LIN {X 0,Y 354.829,Z 449.908,A -85,B 0,C 180,E1 -13477.894,E2 -13477.894} C_VEL
LIN {X 0,Y 354.917,Z 449.897,A -85,B 0,C 180,E1 -13481.892,E2 -13481.892} C_VEL
LIN {X 0,Y 354.937,Z 449.895,A -85,B 0,C 180,E1 -13485.981,E2 -13485.981} C_VEL
LIN {X 0,Y 354.973,Z 449.891,A -85,B 0,C 180,E1 -13489.736,E2 -13489.736} C_VEL
LIN {X 0,Y 355.108,Z 449.874,A -85,B 0,C 180,E1 -13492.037,E2 -13492.037} C_VEL
LIN {X 0,Y 355.087,Z 449.879,A -85,B 0,C 180,E1 -13494.321,E2 -13494.321} C_VEL
LIN {X 0,Y 355.241,Z 449.857,A -85,B 0,C 180,E1 -13497.733,E2 -13497.733} C_VEL
LIN {X 0,Y 355.392,Z 449.839,A -85,B 0,C 180,E1 -13500,E2 -13500} C_VEL
LIN {X 0,Y 355.241,Z 449.86,A -85,B 0,C 180,E1 -13502.268,E2 -13502.268} C_VEL
LIN {X 0,Y 355.137,Z 449.873,A -85,B 0,C 180,E1 -13506.819,E2 -13506.819} C_VEL
LIN {X 0,Y 355.01,Z 449.887,A -85,B 0,C 180,E1 -13509.113,E2 -13509.113} C_VEL
LIN {X 0,Y 354.916,Z 449.902,A -85,B 0,C 180,E1 -13512.581,E2 -13512.581} C_VEL
LIN {X 0,Y 354.884,Z 449.905,A -85,B 0,C 180,E1 -13516.096,E2 -13516.096} C_VEL
LIN {X 0,Y 354.902,Z 449.904,A -85,B 0,C 180,E1 -13518.472,E2 -13518.472} C_VEL
LIN {X 0,Y 354.83,Z 449.912,A -85,B 0,C 180,E1 -13522.107,E2 -13522.107} C_VEL
LIN {X 0,Y 354.895,Z 449.903,A -85,B 0,C 180,E1 -13525.828,E2 -13525.828} C_VEL
LIN {X 0,Y 354.85,Z 449.907,A -85,B 0,C 180,E1 -13529.679,E2 -13529.679} C_VEL
LIN {X 0,Y 354.803,Z 449.914,A -85,B 0,C 180,E1 -13533.703,E2 -13533.703} C_VEL
LIN {X 0,Y 354.796,Z 449.915,A -85,B 0,C 180,E1 -13536.46,E2 -13536.46} C_VEL
LIN {X 0,Y 354.822,Z 449.91,A -85,B 0,C 180,E1 -13539.424,E2 -13539.424} C_VEL
LIN {X 0,Y 354.787,Z 449.914,A -85,B 0,C 180,E1 -13542.868,E2 -13542.868} C_VEL
LIN {X 0,Y 354.775,Z 449.92,A -85,B 0,C 180,E1 -13546.106,E2 -13546.106} C_VEL
LIN {X 0,Y 354.824,Z 449.909,A -85,B 0,C 180,E1 -13549.185,E2 -13549.185} C_VEL
LIN {X 0,Y 354.809,Z 449.913,A -85,B 0,C 180,E1 -13552.403,E2 -13552.403} C_VEL
LIN {X 0,Y 354.813,Z 449.91,A -85,B 0,C 180,E1 -13554.942,E2 -13554.942} C_VEL
LIN {X 0,Y 354.795,Z 449.914,A -85,B 0,C 180,E1 -13558.406,E2 -13558.406} C_VEL
LIN {X 0,Y 354.855,Z 449.91,A -85,B 0,C 180,E1 -13561.62,E2 -13561.62} C_VEL
LIN {X 0,Y 354.901,Z 449.902,A -85,B 0,C 180,E1 -13564.173,E2 -13564.173} C_VEL
LIN {X 0,Y 354.837,Z 449.911,A -85,B 0,C 180,E1 -13567.895,E2 -13567.895} C_VEL
LIN {X 0,Y 354.926,Z 449.9,A -85,B 0,C 180,E1 -13571.892,E2 -13571.892} C_VEL
LIN {X 0,Y 354.946,Z 449.896,A -85,B 0,C 180,E1 -13575.981,E2 -13575.981} C_VEL
LIN {X 0,Y 354.981,Z 449.894,A -85,B 0,C 180,E1 -13579.736,E2 -13579.736} C_VEL
LIN {X 0,Y 355.103,Z 449.878,A -85,B 0,C 180,E1 -13583.18,E2 -13583.18} C_VEL
LIN {X 0,Y 355.249,Z 449.859,A -85,B 0,C 180,E1 -13587.732,E2 -13587.732} C_VEL
LIN {X 0,Y 355.4,Z 449.838,A -85,B 0,C 180,E1 -13590,E2 -13590} C_VEL
LIN {X 0,Y 355.248,Z 449.857,A -85,B 0,C 180,E1 -13592.268,E2 -13592.268} C_VEL
LIN {X 0,Y 355.126,Z 449.873,A -85,B 0,C 180,E1 -13596.819,E2 -13596.819} C_VEL
LIN {X 0,Y 354.981,Z 449.889,A -85,B 0,C 180,E1 -13600.264,E2 -13600.264} C_VEL
LIN {X 0,Y 354.946,Z 449.894,A -85,B 0,C 180,E1 -13604.019,E2 -13604.019} C_VEL
LIN {X 0,Y 354.925,Z 449.896,A -85,B 0,C 180,E1 -13608.108,E2 -13608.108} C_VEL
LIN {X 0,Y 354.837,Z 449.907,A -85,B 0,C 180,E1 -13612.105,E2 -13612.105} C_VEL
LIN {X 0,Y 354.901,Z 449.9,A -85,B 0,C 180,E1 -13615.827,E2 -13615.827} C_VEL
LIN {X 0,Y 354.855,Z 449.906,A -85,B 0,C 180,E1 -13619.678,E2 -13619.678} C_VEL
LIN {X 0,Y 354.779,Z 449.915,A -85,B 0,C 180,E1 -13623.695,E2 -13623.695} C_VEL
LIN {X 0,Y 354.538,Z 449.947,A -85,B 0,C 180,E1 -13626.49,E2 -13626.49} C_VEL
LIN {X 0,Y 354.177,Z 449.995,A -85,B 0,C 180,E1 -13629.418,E2 -13629.418} C_VEL
LIN {X 0,Y 353.996,Z 450.018,A -85,B 0,C 180,E1 -13631.024,E2 -13631.024} C_VEL
LIN {X 0,Y 353.844,Z 450.744,A -85,B 0,C 180,E1 -13632.702,E2 -13632.702} C_VEL
LIN {X 0,Y 353.757,Z 453.469,A -85,B 0,C 180,E1 -13635.946,E2 -13635.946} C_VEL
LIN {X 0,Y 353.742,Z 455.553,A -85,B 0,C 180,E1 -13638.16,E2 -13638.16} C_VEL
LIN {X 0,Y 358.097,Z 470.69,A -85,B 0,C 180,E1 -13639.011,E2 -13639.011} C_VEL
LIN {X 0,Y 361.351,Z 483.198,A -85,B 0,C 180,E1 -13639.883,E2 -13639.883} C_VEL
LIN {X 0,Y 361.484,Z 485.632,A -85,B 0,C 180,E1 -13640.044,E2 -13640.044} C_VEL
LIN {X 0,Y 360.572,Z 489.26,A -85,B 0,C 180,E1 -13640.246,E2 -13640.246} C_VEL
LIN {X 0,Y 355.882,Z 498.667,A -85,B 0,C 180,E1 -13640.734,E2 -13640.734} C_VEL
LIN {X 0,Y 354.987,Z 502.273,A -85,B 0,C 180,E1 -13641.006,E2 -13641.006} C_VEL
LIN {X 0,Y 353.73,Z 515.023,A -85,B 0,C 180,E1 -13642.22,E2 -13642.22} C_VEL
LIN {X 0,Y 352.398,Z 526.861,A -85,B 0,C 180,E1 -13643.607,E2 -13643.607} C_VEL
LIN {X 0,Y 351.136,Z 537.648,A -85,B 0,C 180,E1 -13645.145,E2 -13645.145} C_VEL
LIN {X 0,Y 349.979,Z 547.411,A -85,B 0,C 180,E1 -13646.824,E2 -13646.824} C_VEL
LIN {X 0,Y 348.764,Z 556.624,A -85,B 0,C 180,E1 -13648.742,E2 -13648.742} C_VEL
LIN {X 0,Y 347.986,Z 563.988,A -85,B 0,C 180,E1 -13650.618,E2 -13650.618} C_VEL
LIN {X 0,Y 347.432,Z 569.383,A -85,B 0,C 180,E1 -13652.273,E2 -13652.273} C_VEL
LIN {X 0,Y 346.933,Z 574.46,A -85,B 0,C 180,E1 -13654.18,E2 -13654.18} C_VEL
LIN {X 0,Y 346.575,Z 578.385,A -85,B 0,C 180,E1 -13656.073,E2 -13656.073} C_VEL
LIN {X 0,Y 346.371,Z 580.441,A -85,B 0,C 180,E1 -13657.324,E2 -13657.324} C_VEL
LIN {X 0,Y 346.25,Z 582.506,A -85,B 0,C 180,E1 -13659.014,E2 -13659.014} C_VEL
LIN {X 0,Y 346.14,Z 584.057,A -85,B 0,C 180,E1 -13661.042,E2 -13661.042} C_VEL
LIN {X 0,Y 346.193,Z 584.56,A -85,B 0,C 180,E1 -13662.577,E2 -13662.577} C_VEL
LIN {X 0,Y 346.282,Z 584.255,A -85,B 0,C 180,E1 -13664.701,E2 -13664.701} C_VEL
LIN {X 0,Y 346.641,Z 582.569,A -85,B 0,C 180,E1 -13667.113,E2 -13667.113} C_VEL
LIN {X 0,Y 347.177,Z 579.418,A -85,B 0,C 180,E1 -13669.502,E2 -13669.502} C_VEL
LIN {X 0,Y 347.95,Z 574.76,A -85,B 0,C 180,E1 -13671.872,E2 -13671.872} C_VEL
LIN {X 0,Y 349.05,Z 568.481,A -85,B 0,C 180,E1 -13674.222,E2 -13674.222} C_VEL
LIN {X 0,Y 350.323,Z 561.496,A -85,B 0,C 180,E1 -13676.261,E2 -13676.261} C_VEL
LIN {X 0,Y 351.606,Z 554.204,A -85,B 0,C 180,E1 -13678.007,E2 -13678.007} C_VEL
LIN {X 0,Y 353.21,Z 545.579,A -85,B 0,C 180,E1 -13679.715,E2 -13679.715} C_VEL
LIN {X 0,Y 355.07,Z 535.172,A -85,B 0,C 180,E1 -13681.418,E2 -13681.418} C_VEL
LIN {X 0,Y 356.945,Z 523.616,A -85,B 0,C 180,E1 -13682.962,E2 -13682.962} C_VEL
LIN {X 0,Y 358.844,Z 510.865,A -85,B 0,C 180,E1 -13684.352,E2 -13684.352} C_VEL
LIN {X 0,Y 360.62,Z 497.644,A -85,B 0,C 180,E1 -13685.503,E2 -13685.503} C_VEL
LIN {X 0,Y 360.499,Z 495.401,A -85,B 0,C 180,E1 -13685.715,E2 -13685.715} C_VEL
LIN {X 0,Y 356.948,Z 482.251,A -85,B 0,C 180,E1 -13687.113,E2 -13687.113} C_VEL
LIN {X 0,Y 352.491,Z 471.337,A -85,B 0,C 180,E1 -13688.319,E2 -13688.319} C_VEL
LIN {X 0,Y 349.273,Z 464.852,A -85,B 0,C 180,E1 -13689.061,E2 -13689.061} C_VEL
LIN {X 0,Y 348.009,Z 462.121,A -85,B 0,C 180,E1 -13689.352,E2 -13689.352} C_VEL
LIN {X 0,Y 347.894,Z 461.481,A -85,B 0,C 180,E1 -13689.447,E2 -13689.447} C_VEL
LIN {X 0,Y 348.089,Z 459.823,A -85,B 0,C 180,E1 -13692.832,E2 -13692.832} C_VEL
LIN {X 0,Y 348.261,Z 458.785,A -85,B 0,C 180,E1 -13695.209,E2 -13695.209} C_VEL
LIN {X 0,Y 348.561,Z 457.476,A -85,B 0,C 180,E1 -13698.82,E2 -13698.82} C_VEL
LIN {X 0,Y 348.633,Z 456.533,A -85,B 0,C 180,E1 -13702.52,E2 -13702.52} C_VEL
LIN {X 0,Y 348.681,Z 456.169,A -85,B 0,C 180,E1 -13705.041,E2 -13705.041} C_VEL
LIN {X 0,Y 348.679,Z 456.038,A -85,B 0,C 180,E1 -13707.619,E2 -13707.619} C_VEL
LIN {X 0,Y 348.7,Z 456.207,A -85,B 0,C 180,E1 -13710.256,E2 -13710.256} C_VEL
LIN {X 0,Y 348.809,Z 456.707,A -85,B 0,C 180,E1 -13712.957,E2 -13712.957} C_VEL
LIN {X 0,Y 348.995,Z 457.843,A -85,B 0,C 180,E1 -13716.342,E2 -13716.342} C_VEL
LIN {X 0,Y 349.394,Z 459.832,A -85,B 0,C 180,E1 -13720.151,E2 -13720.151} C_VEL
LIN {X 0,Y 349.843,Z 462.423,A -85,B 0,C 180,E1 -13723.681,E2 -13723.681} C_VEL
LIN {X 0,Y 350.325,Z 465.525,A -85,B 0,C 180,E1 -13726.994,E2 -13726.994} C_VEL
LIN {X 0,Y 350.645,Z 468.414,A -85,B 0,C 180,E1 -13729.608,E2 -13729.608} C_VEL
LIN {X 0,Y 350.514,Z 470.912,A -85,B 0,C 180,E1 -13731.57,E2 -13731.57} C_VEL
LIN {X 0,Y 349.85,Z 474.877,A -85,B 0,C 180,E1 -13734.369,E2 -13734.369} C_VEL
LIN {X 0,Y 349.012,Z 480.13,A -85,B 0,C 180,E1 -13737.752,E2 -13737.752} C_VEL
LIN {X 0,Y 348.283,Z 485.659,A -85,B 0,C 180,E1 -13741.034,E2 -13741.034} C_VEL
LIN {X 0,Y 347.988,Z 488.32,A -85,B 0,C 180,E1 -13742.549,E2 -13742.549} C_VEL
LIN {X 0,Y 348.94,Z 491.893,A -85,B 0,C 180,E1 -13742.833,E2 -13742.833} C_VEL
LIN {X 0,Y 352.14,Z 502.047,A -85,B 0,C 180,E1 -13743.686,E2 -13743.686} C_VEL
LIN {X 0,Y 355.247,Z 515.449,A -85,B 0,C 180,E1 -13744.835,E2 -13744.835} C_VEL
LIN {X 0,Y 356.989,Z 529.251,A -85,B 0,C 180,E1 -13746.039,E2 -13746.039} C_VEL
LIN {X 0,Y 357.339,Z 542.457,A -85,B 0,C 180,E1 -13747.296,E2 -13747.296} C_VEL
LIN {X 0,Y 355.2,Z 556.001,A -85,B 0,C 180,E1 -13748.646,E2 -13748.646} C_VEL
LIN {X 0,Y 353.175,Z 568.787,A -85,B 0,C 180,E1 -13750.228,E2 -13750.228} C_VEL
LIN {X 0,Y 351.295,Z 580.082,A -85,B 0,C 180,E1 -13751.936,E2 -13751.936} C_VEL
LIN {X 0,Y 349.771,Z 589.495,A -85,B 0,C 180,E1 -13753.662,E2 -13753.662} C_VEL
LIN {X 0,Y 348.467,Z 598.551,A -85,B 0,C 180,E1 -13755.672,E2 -13755.672} C_VEL
LIN {X 0,Y 347.475,Z 606.146,A -85,B 0,C 180,E1 -13757.739,E2 -13757.739} C_VEL
LIN {X 0,Y 346.705,Z 612.966,A -85,B 0,C 180,E1 -13760.078,E2 -13760.078} C_VEL
LIN {X 0,Y 346.371,Z 618.146,A -85,B 0,C 180,E1 -13762.421,E2 -13762.421} C_VEL
LIN {X 0,Y 346.248,Z 621.01,A -85,B 0,C 180,E1 -13764.175,E2 -13764.175} C_VEL
LIN {X 0,Y 346.219,Z 623.573,A -85,B 0,C 180,E1 -13766.509,E2 -13766.509} C_VEL
LIN {X 0,Y 346.4,Z 624.733,A -85,B 0,C 180,E1 -13768.837,E2 -13768.837} C_VEL
LIN {X 0,Y 346.41,Z 624.472,A -85,B 0,C 180,E1 -13771.162,E2 -13771.162} C_VEL
LIN {X 0,Y 346.231,Z 622.778,A -85,B 0,C 180,E1 -13773.491,E2 -13773.491} C_VEL
LIN {X 0,Y 346.3,Z 621.398,A -85,B 0,C 180,E1 -13774.656,E2 -13774.656} C_VEL
LIN {X 0,Y 346.366,Z 617.463,A -85,B 0,C 180,E1 -13776.993,E2 -13776.993} C_VEL
LIN {X 0,Y 346.609,Z 611.869,A -85,B 0,C 180,E1 -13779.335,E2 -13779.335} C_VEL
LIN {X 0,Y 347.095,Z 605.516,A -85,B 0,C 180,E1 -13781.386,E2 -13781.386} C_VEL
LIN {X 0,Y 347.902,Z 597.587,A -85,B 0,C 180,E1 -13783.433,E2 -13783.433} C_VEL
LIN {X 0,Y 348.598,Z 590.314,A -85,B 0,C 180,E1 -13784.988,E2 -13784.988} C_VEL
LIN {X 0,Y 349.659,Z 581.104,A -85,B 0,C 180,E1 -13786.643,E2 -13786.643} C_VEL
LIN {X 0,Y 350.922,Z 570.429,A -85,B 0,C 180,E1 -13788.235,E2 -13788.235} C_VEL
LIN {X 0,Y 352.268,Z 560.02,A -85,B 0,C 180,E1 -13789.522,E2 -13789.522} C_VEL
LIN {X 0,Y 353.719,Z 547.45,A -85,B 0,C 180,E1 -13790.803,E2 -13790.803} C_VEL
LIN {X 0,Y 354.551,Z 539.176,A -85,B 0,C 180,E1 -13791.512,E2 -13791.512} C_VEL
LIN {X 0,Y 353.044,Z 526.06,A -85,B 0,C 180,E1 -13792.554,E2 -13792.554} C_VEL
LIN {X 0,Y 350.623,Z 511.086,A -85,B 0,C 180,E1 -13793.529,E2 -13793.529} C_VEL
LIN {X 0,Y 347.827,Z 495.803,A -85,B 0,C 180,E1 -13794.297,E2 -13794.297} C_VEL
LIN {X 0,Y 347.476,Z 493.605,A -85,B 0,C 180,E1 -13794.412,E2 -13794.412} C_VEL
LIN {X 0,Y 348.026,Z 487.442,A -85,B 0,C 180,E1 -13797.675,E2 -13797.675} C_VEL
LIN {X 0,Y 348.651,Z 481.404,A -85,B 0,C 180,E1 -13800.931,E2 -13800.931} C_VEL
LIN {X 0,Y 349.401,Z 475.058,A -85,B 0,C 180,E1 -13804.443,E2 -13804.443} C_VEL
LIN {X 0,Y 350.106,Z 469.257,A -85,B 0,C 180,E1 -13807.752,E2 -13807.752} C_VEL
LIN {X 0,Y 350.303,Z 465.561,A -85,B 0,C 180,E1 -13809.941,E2 -13809.941} C_VEL
LIN {X 0,Y 349.553,Z 460.534,A -85,B 0,C 180,E1 -13813.124,E2 -13813.124} C_VEL
LIN {X 0,Y 348.571,Z 455.182,A -85,B 0,C 180,E1 -13816.724,E2 -13816.724} C_VEL
LIN {X 0,Y 347.827,Z 450.784,A -85,B 0,C 180,E1 -13819.854,E2 -13819.854} C_VEL
LIN {X 0,Y 347.766,Z 450.788,A -85,B 0,C 180,E1 -13823.935,E2 -13823.935} C_VEL
LIN {X 0,Y 347.743,Z 450.796,A -85,B 0,C 180,E1 -13826.929,E2 -13826.929} C_VEL
LIN {X 0,Y 347.802,Z 450.789,A -85,B 0,C 180,E1 -13830.99,E2 -13830.99} C_VEL
LIN {X 0,Y 347.827,Z 450.781,A -85,B 0,C 180,E1 -13833.608,E2 -13833.608} C_VEL
LIN {X 0,Y 347.783,Z 450.786,A -85,B 0,C 180,E1 -13836.162,E2 -13836.162} C_VEL
LIN {X 0,Y 347.807,Z 450.783,A -85,B 0,C 180,E1 -13839.909,E2 -13839.909} C_VEL
LIN {X 0,Y 347.861,Z 450.778,A -85,B 0,C 180,E1 -13842.359,E2 -13842.359} C_VEL
LIN {X 0,Y 347.892,Z 450.772,A -85,B 0,C 180,E1 -13845.971,E2 -13845.971} C_VEL
LIN {X 0,Y 347.923,Z 450.769,A -85,B 0,C 180,E1 -13849.526,E2 -13849.526} C_VEL
LIN {X 0,Y 348.068,Z 450.751,A -85,B 0,C 180,E1 -13851.875,E2 -13851.875} C_VEL
LIN {X 0,Y 348.062,Z 450.753,A -85,B 0,C 180,E1 -13854.206,E2 -13854.206} C_VEL
LIN {X 0,Y 348.203,Z 450.734,A -85,B 0,C 180,E1 -13857.687,E2 -13857.687} C_VEL
LIN {X 0,Y 348.34,Z 450.717,A -85,B 0,C 180,E1 -13860,E2 -13860} C_VEL
LIN {X 0,Y 348.203,Z 450.737,A -85,B 0,C 180,E1 -13862.314,E2 -13862.314} C_VEL
LIN {X 0,Y 348.104,Z 450.748,A -85,B 0,C 180,E1 -13866.958,E2 -13866.958} C_VEL
LIN {X 0,Y 347.962,Z 450.764,A -85,B 0,C 180,E1 -13869.299,E2 -13869.299} C_VEL
LIN {X 0,Y 347.885,Z 450.775,A -85,B 0,C 180,E1 -13872.84,E2 -13872.84} C_VEL
LIN {X 0,Y 347.834,Z 450.785,A -85,B 0,C 180,E1 -13876.432,E2 -13876.432} C_VEL
LIN {X 0,Y 347.851,Z 450.779,A -85,B 0,C 180,E1 -13878.861,E2 -13878.861} C_VEL
LIN {X 0,Y 347.77,Z 450.791,A -85,B 0,C 180,E1 -13882.58,E2 -13882.58} C_VEL
LIN {X 0,Y 347.808,Z 450.783,A -85,B 0,C 180,E1 -13885.109,E2 -13885.109} C_VEL
LIN {X 0,Y 347.806,Z 450.784,A -85,B 0,C 180,E1 -13887.695,E2 -13887.695} C_VEL
LIN {X 0,Y 347.76,Z 450.793,A -85,B 0,C 180,E1 -13890.347,E2 -13890.347} C_VEL
LIN {X 0,Y 347.741,Z 450.794,A -85,B 0,C 180,E1 -13894.465,E2 -13894.465} C_VEL
LIN {X 0,Y 347.772,Z 450.793,A -85,B 0,C 180,E1 -13897.99,E2 -13897.99} C_VEL
LIN {X 0,Y 347.749,Z 450.794,A -85,B 0,C 180,E1 -13901.831,E2 -13901.831} C_VEL
LIN {X 0,Y 347.707,Z 450.795,A -85,B 0,C 180,E1 -13905.027,E2 -13905.027} C_VEL
LIN {X 0,Y 347.767,Z 450.79,A -85,B 0,C 180,E1 -13908.395,E2 -13908.395} C_VEL
LIN {X 0,Y 347.776,Z 450.792,A -85,B 0,C 180,E1 -13912.012,E2 -13912.012} C_VEL
LIN {X 0,Y 347.745,Z 450.794,A -85,B 0,C 180,E1 -13915.537,E2 -13915.537} C_VEL
LIN {X 0,Y 347.765,Z 450.793,A -85,B 0,C 180,E1 -13919.654,E2 -13919.654} C_VEL
LIN {X 0,Y 347.854,Z 450.777,A -85,B 0,C 180,E1 -13922.745,E2 -13922.745} C_VEL
LIN {X 0,Y 347.791,Z 450.787,A -85,B 0,C 180,E1 -13926.163,E2 -13926.163} C_VEL
LIN {X 0,Y 347.82,Z 450.785,A -85,B 0,C 180,E1 -13929.91,E2 -13929.91} C_VEL
LIN {X 0,Y 347.869,Z 450.776,A -85,B 0,C 180,E1 -13932.36,E2 -13932.36} C_VEL
LIN {X 0,Y 347.9,Z 450.773,A -85,B 0,C 180,E1 -13935.971,E2 -13935.971} C_VEL
LIN {X 0,Y 347.932,Z 450.773,A -85,B 0,C 180,E1 -13939.526,E2 -13939.526} C_VEL
LIN {X 0,Y 348.071,Z 450.752,A -85,B 0,C 180,E1 -13943.042,E2 -13943.042} C_VEL
LIN {X 0,Y 348.211,Z 450.736,A -85,B 0,C 180,E1 -13947.687,E2 -13947.687} C_VEL
LIN {X 0,Y 348.349,Z 450.716,A -85,B 0,C 180,E1 -13950,E2 -13950} C_VEL
LIN {X 0,Y 348.21,Z 450.733,A -85,B 0,C 180,E1 -13952.313,E2 -13952.313} C_VEL
LIN {X 0,Y 348.092,Z 450.75,A -85,B 0,C 180,E1 -13956.958,E2 -13956.958} C_VEL
LIN {X 0,Y 347.932,Z 450.768,A -85,B 0,C 180,E1 -13960.474,E2 -13960.474} C_VEL
LIN {X 0,Y 347.901,Z 450.771,A -85,B 0,C 180,E1 -13964.149,E2 -13964.149} C_VEL
LIN {X 0,Y 347.893,Z 450.772,A -85,B 0,C 180,E1 -13968.29,E2 -13968.29} C_VEL
LIN {X 0,Y 347.791,Z 450.786,A -85,B 0,C 180,E1 -13971.635,E2 -13971.635} C_VEL
LIN {X 0,Y 347.815,Z 450.787,A -85,B 0,C 180,E1 -13975.108,E2 -13975.108} C_VEL
LIN {X 0,Y 347.811,Z 450.783,A -85,B 0,C 180,E1 -13977.693,E2 -13977.693} C_VEL
LIN {X 0,Y 347.764,Z 450.789,A -85,B 0,C 180,E1 -13980.346,E2 -13980.346} C_VEL
LIN {X 0,Y 347.712,Z 450.795,A -85,B 0,C 180,E1 -13984.034,E2 -13984.034} C_VEL
LIN {X 0,Y 347.383,Z 450.838,A -85,B 0,C 180,E1 -13987.368,E2 -13987.368} C_VEL
LIN {X 0,Y 347.013,Z 450.888,A -85,B 0,C 180,E1 -13990.397,E2 -13990.397} C_VEL
LIN {X 0,Y 346.799,Z 450.914,A -85,B 0,C 180,E1 -13991.97,E2 -13991.97} C_VEL
LIN {X 0,Y 346.719,Z 453.556,A -85,B 0,C 180,E1 -13995.189,E2 -13995.189} C_VEL
LIN {X 0,Y 346.668,Z 455.811,A -85,B 0,C 180,E1 -13997.751,E2 -13997.751} C_VEL
LIN {X 0,Y 350.723,Z 469.912,A -85,B 0,C 180,E1 -13998.56,E2 -13998.56} C_VEL
LIN {X 0,Y 354.542,Z 484.531,A -85,B 0,C 180,E1 -13999.604,E2 -13999.604} C_VEL
LIN {X 0,Y 355.941,Z 491.589,A -85,B 0,C 180,E1 -14000.172,E2 -14000.172} C_VEL
LIN {X 0,Y 354.987,Z 502.273,A -85,B 0,C 180,E1 -14001.006,E2 -14001.006} C_VEL
LIN {X 0,Y 353.88,Z 507.456,A -85,B 0,C 180,E1 -14001.429,E2 -14001.429} C_VEL
LIN {X 0,Y 350.294,Z 515.693,A -85,B 0,C 180,E1 -14002.113,E2 -14002.113} C_VEL
LIN {X 0,Y 346.615,Z 523.574,A -85,B 0,C 180,E1 -14002.897,E2 -14002.897} C_VEL
LIN {X 0,Y 345.377,Z 528.2,A -85,B 0,C 180,E1 -14003.471,E2 -14003.471} C_VEL
LIN {X 0,Y 344.049,Z 539.278,A -85,B 0,C 180,E1 -14005.112,E2 -14005.112} C_VEL
LIN {X 0,Y 342.845,Z 549.219,A -85,B 0,C 180,E1 -14006.898,E2 -14006.898} C_VEL
LIN {X 0,Y 341.687,Z 557.596,A -85,B 0,C 180,E1 -14008.711,E2 -14008.711} C_VEL
LIN {X 0,Y 340.884,Z 565.063,A -85,B 0,C 180,E1 -14010.682,E2 -14010.682} C_VEL
LIN {X 0,Y 340.128,Z 571.996,A -85,B 0,C 180,E1 -14012.962,E2 -14012.962} C_VEL
LIN {X 0,Y 339.709,Z 576.583,A -85,B 0,C 180,E1 -14014.905,E2 -14014.905} C_VEL
LIN {X 0,Y 339.349,Z 580.082,A -85,B 0,C 180,E1 -14016.828,E2 -14016.828} C_VEL
LIN {X 0,Y 339.174,Z 582.694,A -85,B 0,C 180,E1 -14018.816,E2 -14018.816} C_VEL
LIN {X 0,Y 339.079,Z 584.251,A -85,B 0,C 180,E1 -14020.632,E2 -14020.632} C_VEL
LIN {X 0,Y 339.101,Z 585.029,A -85,B 0,C 180,E1 -14023.132,E2 -14023.132} C_VEL
LIN {X 0,Y 339.319,Z 584.338,A -85,B 0,C 180,E1 -14025.608,E2 -14025.608} C_VEL
LIN {X 0,Y 339.743,Z 582.218,A -85,B 0,C 180,E1 -14028.061,E2 -14028.061} C_VEL
LIN {X 0,Y 340.421,Z 578.652,A -85,B 0,C 180,E1 -14030.493,E2 -14030.493} C_VEL
LIN {X 0,Y 341.086,Z 574.873,A -85,B 0,C 180,E1 -14032.338,E2 -14032.338} C_VEL
LIN {X 0,Y 342.308,Z 568.637,A -85,B 0,C 180,E1 -14034.699,E2 -14034.699} C_VEL
LIN {X 0,Y 343.717,Z 561.604,A -85,B 0,C 180,E1 -14036.776,E2 -14036.776} C_VEL
LIN {X 0,Y 345.32,Z 552.941,A -85,B 0,C 180,E1 -14038.834,E2 -14038.834} C_VEL
LIN {X 0,Y 347.108,Z 543.891,A -85,B 0,C 180,E1 -14040.58,E2 -14040.58} C_VEL
LIN {X 0,Y 349.117,Z 533.081,A -85,B 0,C 180,E1 -14042.307,E2 -14042.307} C_VEL
LIN {X 0,Y 351.19,Z 521.065,A -85,B 0,C 180,E1 -14043.873,E2 -14043.873} C_VEL
LIN {X 0,Y 353.203,Z 508.147,A -85,B 0,C 180,E1 -14045.23,E2 -14045.23} C_VEL
LIN {X 0,Y 354.445,Z 498.262,A -85,B 0,C 180,E1 -14046.088,E2 -14046.088} C_VEL
LIN {X 0,Y 351.256,Z 485.636,A -85,B 0,C 180,E1 -14047.523,E2 -14047.523} C_VEL
LIN {X 0,Y 346.264,Z 473.099,A -85,B 0,C 180,E1 -14049,E2 -14049} C_VEL
LIN {X 0,Y 342.347,Z 465.595,A -85,B 0,C 180,E1 -14049.94,E2 -14049.94} C_VEL
LIN {X 0,Y 341.095,Z 462.937,A -85,B 0,C 180,E1 -14050.248,E2 -14050.248} C_VEL
LIN {X 0,Y 340.973,Z 462.196,A -85,B 0,C 180,E1 -14050.352,E2 -14050.352} C_VEL
LIN {X 0,Y 341.251,Z 460.309,A -85,B 0,C 180,E1 -14054.548,E2 -14054.548} C_VEL
LIN {X 0,Y 341.607,Z 458.778,A -85,B 0,C 180,E1 -14058.852,E2 -14058.852} C_VEL
LIN {X 0,Y 341.683,Z 457.983,A -85,B 0,C 180,E1 -14062.244,E2 -14062.244} C_VEL
LIN {X 0,Y 341.711,Z 457.556,A -85,B 0,C 180,E1 -14065.589,E2 -14065.589} C_VEL
LIN {X 0,Y 341.714,Z 457.546,A -85,B 0,C 180,E1 -14068.232,E2 -14068.232} C_VEL
LIN {X 0,Y 341.762,Z 457.817,A -85,B 0,C 180,E1 -14070.937,E2 -14070.937} C_VEL
LIN {X 0,Y 341.878,Z 458.436,A -85,B 0,C 180,E1 -14073.713,E2 -14073.713} C_VEL
LIN {X 0,Y 342.1,Z 459.568,A -85,B 0,C 180,E1 -14076.756,E2 -14076.756} C_VEL
LIN {X 0,Y 342.385,Z 460.999,A -85,B 0,C 180,E1 -14079.518,E2 -14079.518} C_VEL
LIN {X 0,Y 342.772,Z 463.057,A -85,B 0,C 180,E1 -14082.579,E2 -14082.579} C_VEL
LIN {X 0,Y 343.214,Z 465.864,A -85,B 0,C 180,E1 -14085.877,E2 -14085.877} C_VEL
LIN {X 0,Y 343.474,Z 467.495,A -85,B 0,C 180,E1 -14087.529,E2 -14087.529} C_VEL
LIN {X 0,Y 343.636,Z 469.296,A -85,B 0,C 180,E1 -14089.176,E2 -14089.176} C_VEL
LIN {X 0,Y 343.405,Z 472.97,A -85,B 0,C 180,E1 -14092.124,E2 -14092.124} C_VEL
LIN {X 0,Y 342.658,Z 477.228,A -85,B 0,C 180,E1 -14095.126,E2 -14095.126} C_VEL
LIN {X 0,Y 341.713,Z 483.346,A -85,B 0,C 180,E1 -14099.058,E2 -14099.058} C_VEL
LIN {X 0,Y 341.159,Z 487.68,A -85,B 0,C 180,E1 -14101.656,E2 -14101.656} C_VEL
LIN {X 0,Y 342.044,Z 491.064,A -85,B 0,C 180,E1 -14101.929,E2 -14101.929} C_VEL
LIN {X 0,Y 345.422,Z 501.575,A -85,B 0,C 180,E1 -14102.895,E2 -14102.895} C_VEL
LIN {X 0,Y 348.64,Z 514.814,A -85,B 0,C 180,E1 -14104.102,E2 -14104.102} C_VEL
LIN {X 0,Y 350.333,Z 527.227,A -85,B 0,C 180,E1 -14105.253,E2 -14105.253} C_VEL
LIN {X 0,Y 350.875,Z 538.928,A -85,B 0,C 180,E1 -14106.385,E2 -14106.385} C_VEL
LIN {X 0,Y 350.632,Z 544.943,A -85,B 0,C 180,E1 -14106.993,E2 -14106.993} C_VEL
LIN {X 0,Y 348.605,Z 556.949,A -85,B 0,C 180,E1 -14108.256,E2 -14108.256} C_VEL
LIN {X 0,Y 346.508,Z 569.173,A -85,B 0,C 180,E1 -14109.831,E2 -14109.831} C_VEL
LIN {X 0,Y 344.547,Z 580.283,A -85,B 0,C 180,E1 -14111.569,E2 -14111.569} C_VEL
LIN {X 0,Y 342.935,Z 589.588,A -85,B 0,C 180,E1 -14113.327,E2 -14113.327} C_VEL
LIN {X 0,Y 341.565,Z 598.046,A -85,B 0,C 180,E1 -14115.255,E2 -14115.255} C_VEL
LIN {X 0,Y 340.491,Z 606.005,A -85,B 0,C 180,E1 -14117.483,E2 -14117.483} C_VEL
LIN {X 0,Y 339.658,Z 612.769,A -85,B 0,C 180,E1 -14119.871,E2 -14119.871} C_VEL
LIN {X 0,Y 339.292,Z 617.889,A -85,B 0,C 180,E1 -14122.262,E2 -14122.262} C_VEL
LIN {X 0,Y 339.169,Z 620.688,A -85,B 0,C 180,E1 -14124.053,E2 -14124.053} C_VEL
LIN {X 0,Y 339.14,Z 623.201,A -85,B 0,C 180,E1 -14126.436,E2 -14126.436} C_VEL
LIN {X 0,Y 339.317,Z 624.315,A -85,B 0,C 180,E1 -14128.813,E2 -14128.813} C_VEL
LIN {X 0,Y 339.347,Z 624.005,A -85,B 0,C 180,E1 -14131.187,E2 -14131.187} C_VEL
LIN {X 0,Y 339.155,Z 622.255,A -85,B 0,C 180,E1 -14133.564,E2 -14133.564} C_VEL
LIN {X 0,Y 339.212,Z 620.838,A -85,B 0,C 180,E1 -14134.754,E2 -14134.754} C_VEL
LIN {X 0,Y 339.304,Z 616.816,A -85,B 0,C 180,E1 -14137.139,E2 -14137.139} C_VEL
LIN {X 0,Y 339.549,Z 611.15,A -85,B 0,C 180,E1 -14139.531,E2 -14139.531} C_VEL
LIN {X 0,Y 340.102,Z 604.724,A -85,B 0,C 180,E1 -14141.623,E2 -14141.623} C_VEL
LIN {X 0,Y 340.86,Z 596.698,A -85,B 0,C 180,E1 -14143.716,E2 -14143.716} C_VEL
LIN {X 0,Y 341.772,Z 588.304,A -85,B 0,C 180,E1 -14145.505,E2 -14145.505} C_VEL
LIN {X 0,Y 343.045,Z 578.24,A -85,B 0,C 180,E1 -14147.281,E2 -14147.281} C_VEL
LIN {X 0,Y 344.415,Z 567.059,A -85,B 0,C 180,E1 -14148.901,E2 -14148.901} C_VEL
LIN {X 0,Y 345.782,Z 556.069,A -85,B 0,C 180,E1 -14150.213,E2 -14150.213} C_VEL
LIN {X 0,Y 347.127,Z 544.291,A -85,B 0,C 180,E1 -14151.372,E2 -14151.372} C_VEL
LIN {X 0,Y 347.587,Z 539.195,A -85,B 0,C 180,E1 -14151.81,E2 -14151.81} C_VEL
LIN {X 0,Y 346.031,Z 525.911,A -85,B 0,C 180,E1 -14152.9,E2 -14152.9} C_VEL
LIN {X 0,Y 343.632,Z 511.092,A -85,B 0,C 180,E1 -14153.897,E2 -14153.897} C_VEL
LIN {X 0,Y 340.811,Z 495.483,A -85,B 0,C 180,E1 -14154.709,E2 -14154.709} C_VEL
LIN {X 0,Y 340.473,Z 493.264,A -85,B 0,C 180,E1 -14154.821,E2 -14154.821} C_VEL
LIN {X 0,Y 341.033,Z 486.884,A -85,B 0,C 180,E1 -14158.293,E2 -14158.293} C_VEL
LIN {X 0,Y 341.706,Z 480.87,A -85,B 0,C 180,E1 -14161.632,E2 -14161.632} C_VEL
LIN {X 0,Y 342.46,Z 474.815,A -85,B 0,C 180,E1 -14165.072,E2 -14165.072} C_VEL
LIN {X 0,Y 343.097,Z 469.951,A -85,B 0,C 180,E1 -14167.916,E2 -14167.916} C_VEL
LIN {X 0,Y 343.267,Z 466.447,A -85,B 0,C 180,E1 -14170.045,E2 -14170.045} C_VEL
LIN {X 0,Y 342.503,Z 461.357,A -85,B 0,C 180,E1 -14173.334,E2 -14173.334} C_VEL
LIN {X 0,Y 341.463,Z 455.705,A -85,B 0,C 180,E1 -14177.218,E2 -14177.218} C_VEL
LIN {X 0,Y 340.744,Z 451.666,A -85,B 0,C 180,E1 -14180.254,E2 -14180.254} C_VEL
LIN {X 0,Y 340.706,Z 451.669,A -85,B 0,C 180,E1 -14183.559,E2 -14183.559} C_VEL
LIN {X 0,Y 340.691,Z 451.669,A -85,B 0,C 180,E1 -14186.153,E2 -14186.153} C_VEL
LIN {X 0,Y 340.771,Z 451.66,A -85,B 0,C 180,E1 -14190.332,E2 -14190.332} C_VEL
LIN {X 0,Y 340.8,Z 451.661,A -85,B 0,C 180,E1 -14193.02,E2 -14193.02} C_VEL
LIN {X 0,Y 340.723,Z 451.671,A -85,B 0,C 180,E1 -14196.927,E2 -14196.927} C_VEL
LIN {X 0,Y 340.785,Z 451.662,A -85,B 0,C 180,E1 -14200.733,E2 -14200.733} C_VEL
LIN {X 0,Y 340.781,Z 451.66,A -85,B 0,C 180,E1 -14203.219,E2 -14203.219} C_VEL
LIN {X 0,Y 340.838,Z 451.656,A -85,B 0,C 180,E1 -14206.89,E2 -14206.89} C_VEL
LIN {X 0,Y 340.923,Z 451.644,A -85,B 0,C 180,E1 -14210.508,E2 -14210.508} C_VEL
LIN {X 0,Y 341.07,Z 451.626,A -85,B 0,C 180,E1 -14212.898,E2 -14212.898} C_VEL
LIN {X 0,Y 341.165,Z 451.61,A -85,B 0,C 180,E1 -14217.639,E2 -14217.639} C_VEL
LIN {X 0,Y 341.291,Z 451.595,A -85,B 0,C 180,E1 -14220,E2 -14220} C_VEL
LIN {X 0,Y 341.165,Z 451.614,A -85,B 0,C 180,E1 -14222.361,E2 -14222.361} C_VEL
LIN {X 0,Y 341.073,Z 451.623,A -85,B 0,C 180,E1 -14227.102,E2 -14227.102} C_VEL
LIN {X 0,Y 340.866,Z 451.651,A -85,B 0,C 180,E1 -14230.694,E2 -14230.694} C_VEL
LIN {X 0,Y 340.858,Z 451.653,A -85,B 0,C 180,E1 -14234.325,E2 -14234.325} C_VEL
LIN {X 0,Y 340.833,Z 451.656,A -85,B 0,C 180,E1 -14238.467,E2 -14238.467} C_VEL
LIN {X 0,Y 340.75,Z 451.664,A -85,B 0,C 180,E1 -14241.857,E2 -14241.857} C_VEL
LIN {X 0,Y 340.768,Z 451.661,A -85,B 0,C 180,E1 -14245.665,E2 -14245.665} C_VEL
LIN {X 0,Y 340.737,Z 451.669,A -85,B 0,C 180,E1 -14248.32,E2 -14248.32} C_VEL
LIN {X 0,Y 340.7,Z 451.668,A -85,B 0,C 180,E1 -14251.045,E2 -14251.045} C_VEL
LIN {X 0,Y 340.715,Z 451.666,A -85,B 0,C 180,E1 -14255.28,E2 -14255.28} C_VEL
LIN {X 0,Y 340.708,Z 451.67,A -85,B 0,C 180,E1 -14258.387,E2 -14258.387} C_VEL
LIN {X 0,Y 340.697,Z 451.674,A -85,B 0,C 180,E1 -14262.046,E2 -14262.046} C_VEL
LIN {X 0,Y 340.667,Z 451.676,A -85,B 0,C 180,E1 -14266.225,E2 -14266.225} C_VEL
LIN {X 0,Y 340.703,Z 451.668,A -85,B 0,C 180,E1 -14268.694,E2 -14268.694} C_VEL
LIN {X 0,Y 340.739,Z 451.668,A -85,B 0,C 180,E1 -14271.774,E2 -14271.774} C_VEL
LIN {X 0,Y 340.723,Z 451.669,A -85,B 0,C 180,E1 -14275.596,E2 -14275.596} C_VEL
LIN {X 0,Y 340.705,Z 451.667,A -85,B 0,C 180,E1 -14278.957,E2 -14278.957} C_VEL
LIN {X 0,Y 340.781,Z 451.658,A -85,B 0,C 180,E1 -14282.474,E2 -14282.474} C_VEL
LIN {X 0,Y 340.758,Z 451.666,A -85,B 0,C 180,E1 -14285.639,E2 -14285.639} C_VEL
LIN {X 0,Y 340.751,Z 451.666,A -85,B 0,C 180,E1 -14289.475,E2 -14289.475} C_VEL
LIN {X 0,Y 340.861,Z 451.651,A -85,B 0,C 180,E1 -14291.985,E2 -14291.985} C_VEL
LIN {X 0,Y 340.872,Z 451.651,A -85,B 0,C 180,E1 -14295.705,E2 -14295.705} C_VEL
LIN {X 0,Y 340.874,Z 451.65,A -85,B 0,C 180,E1 -14299.307,E2 -14299.307} C_VEL
LIN {X 0,Y 341.019,Z 451.629,A -85,B 0,C 180,E1 -14302.897,E2 -14302.897} C_VEL
LIN {X 0,Y 341.173,Z 451.613,A -85,B 0,C 180,E1 -14307.639,E2 -14307.639} C_VEL
LIN {X 0,Y 341.299,Z 451.594,A -85,B 0,C 180,E1 -14310,E2 -14310} C_VEL
LIN {X 0,Y 341.172,Z 451.609,A -85,B 0,C 180,E1 -14312.361,E2 -14312.361} C_VEL
LIN {X 0,Y 341.061,Z 451.627,A -85,B 0,C 180,E1 -14317.102,E2 -14317.102} C_VEL
LIN {X 0,Y 340.874,Z 451.648,A -85,B 0,C 180,E1 -14320.693,E2 -14320.693} C_VEL
LIN {X 0,Y 340.866,Z 451.647,A -85,B 0,C 180,E1 -14324.324,E2 -14324.324} C_VEL
LIN {X 0,Y 340.839,Z 451.651,A -85,B 0,C 180,E1 -14328.466,E2 -14328.466} C_VEL
LIN {X 0,Y 340.756,Z 451.661,A -85,B 0,C 180,E1 -14331.856,E2 -14331.856} C_VEL
LIN {X 0,Y 340.774,Z 451.66,A -85,B 0,C 180,E1 -14335.664,E2 -14335.664} C_VEL
LIN {X 0,Y 340.742,Z 451.663,A -85,B 0,C 180,E1 -14338.319,E2 -14338.319} C_VEL
LIN {X 0,Y 340.703,Z 451.673,A -85,B 0,C 180,E1 -14341.044,E2 -14341.044} C_VEL
LIN {X 0,Y 340.64,Z 451.677,A -85,B 0,C 180,E1 -14344.383,E2 -14344.383} C_VEL
LIN {X 0,Y 340.401,Z 451.71,A -85,B 0,C 180,E1 -14346.779,E2 -14346.779} C_VEL
LIN {X 0,Y 339.989,Z 451.764,A -85,B 0,C 180,E1 -14350.107,E2 -14350.107} C_VEL
LIN {X 0,Y 339.77,Z 451.789,A -85,B 0,C 180,E1 -14351.871,E2 -14351.871} C_VEL
LIN {X 0,Y 339.651,Z 454.377,A -85,B 0,C 180,E1 -14355.289,E2 -14355.289} C_VEL
LIN {X 0,Y 339.612,Z 456.076,A -85,B 0,C 180,E1 -14357.311,E2 -14357.311} C_VEL
LIN {X 0,Y 344.38,Z 472.902,A -85,B 0,C 180,E1 -14358.338,E2 -14358.338} C_VEL
LIN {X 0,Y 348.021,Z 487.065,A -85,B 0,C 180,E1 -14359.419,E2 -14359.419} C_VEL
LIN {X 0,Y 349.075,Z 492.952,A -85,B 0,C 180,E1 -14359.911,E2 -14359.911} C_VEL
LIN {X 0,Y 347.834,Z 506.443,A -85,B 0,C 180,E1 -14361.032,E2 -14361.032} C_VEL
LIN {X 0,Y 346.455,Z 518.662,A -85,B 0,C 180,E1 -14362.29,E2 -14362.29} C_VEL
LIN {X 0,Y 345.377,Z 528.2,A -85,B 0,C 180,E1 -14363.471,E2 -14363.471} C_VEL
LIN {X 0,Y 344.174,Z 532.752,A -85,B 0,C 180,E1 -14364.073,E2 -14364.073} C_VEL
LIN {X 0,Y 340.558,Z 539.872,A -85,B 0,C 180,E1 -14365.059,E2 -14365.059} C_VEL
LIN {X 0,Y 336.952,Z 546.615,A -85,B 0,C 180,E1 -14366.128,E2 -14366.128} C_VEL
LIN {X 0,Y 335.762,Z 550.437,A -85,B 0,C 180,E1 -14366.856,E2 -14366.856} C_VEL
LIN {X 0,Y 334.613,Z 558.55,A -85,B 0,C 180,E1 -14368.674,E2 -14368.674} C_VEL
LIN {X 0,Y 333.787,Z 565.934,A -85,B 0,C 180,E1 -14370.689,E2 -14370.689} C_VEL
LIN {X 0,Y 333.033,Z 572.75,A -85,B 0,C 180,E1 -14373.017,E2 -14373.017} C_VEL
LIN {X 0,Y 332.534,Z 577.924,A -85,B 0,C 180,E1 -14375.336,E2 -14375.336} C_VEL
LIN {X 0,Y 332.159,Z 581.635,A -85,B 0,C 180,E1 -14377.613,E2 -14377.613} C_VEL
LIN {X 0,Y 332.094,Z 583.17,A -85,B 0,C 180,E1 -14378.914,E2 -14378.914} C_VEL
LIN {X 0,Y 331.975,Z 585.058,A -85,B 0,C 180,E1 -14381.485,E2 -14381.485} C_VEL
LIN {X 0,Y 332.016,Z 585.434,A -85,B 0,C 180,E1 -14382.761,E2 -14382.761} C_VEL
LIN {X 0,Y 332.205,Z 585.077,A -85,B 0,C 180,E1 -14385.293,E2 -14385.293} C_VEL
LIN {X 0,Y 332.417,Z 584.336,A -85,B 0,C 180,E1 -14386.552,E2 -14386.552} C_VEL
LIN {X 0,Y 332.913,Z 581.776,A -85,B 0,C 180,E1 -14389.047,E2 -14389.047} C_VEL
LIN {X 0,Y 333.721,Z 577.776,A -85,B 0,C 180,E1 -14391.522,E2 -14391.522} C_VEL
LIN {X 0,Y 334.841,Z 572.233,A -85,B 0,C 180,E1 -14393.976,E2 -14393.976} C_VEL
LIN {X 0,Y 335.971,Z 566.92,A -85,B 0,C 180,E1 -14395.801,E2 -14395.801} C_VEL
LIN {X 0,Y 337.559,Z 559.323,A -85,B 0,C 180,E1 -14397.925,E2 -14397.925} C_VEL
LIN {X 0,Y 339.147,Z 551.592,A -85,B 0,C 180,E1 -14399.703,E2 -14399.703} C_VEL
LIN {X 0,Y 341.106,Z 542.251,A -85,B 0,C 180,E1 -14401.476,E2 -14401.476} C_VEL
LIN {X 0,Y 343.302,Z 531.017,A -85,B 0,C 180,E1 -14403.227,E2 -14403.227} C_VEL
LIN {X 0,Y 345.33,Z 519.694,A -85,B 0,C 180,E1 -14404.669,E2 -14404.669} C_VEL
LIN {X 0,Y 347.3,Z 507.513,A -85,B 0,C 180,E1 -14405.942,E2 -14405.942} C_VEL
LIN {X 0,Y 348.266,Z 500.3,A -85,B 0,C 180,E1 -14406.588,E2 -14406.588} C_VEL
LIN {X 0,Y 345.299,Z 488.162,A -85,B 0,C 180,E1 -14408.037,E2 -14408.037} C_VEL
LIN {X 0,Y 340.667,Z 476.514,A -85,B 0,C 180,E1 -14409.518,E2 -14409.518} C_VEL
LIN {X 0,Y 335.818,Z 466.819,A -85,B 0,C 180,E1 -14410.826,E2 -14410.826} C_VEL
LIN {X 0,Y 334.308,Z 464.188,A -85,B 0,C 180,E1 -14411.194,E2 -14411.194} C_VEL
LIN {X 0,Y 334.022,Z 462.938,A -85,B 0,C 180,E1 -14411.338,E2 -14411.338} C_VEL
LIN {X 0,Y 334.281,Z 461.516,A -85,B 0,C 180,E1 -14414.739,E2 -14414.739} C_VEL
LIN {X 0,Y 334.555,Z 460.269,A -85,B 0,C 180,E1 -14418.367,E2 -14418.367} C_VEL
LIN {X 0,Y 334.67,Z 459.628,A -85,B 0,C 180,E1 -14420.916,E2 -14420.916} C_VEL
LIN {X 0,Y 334.782,Z 459.049,A -85,B 0,C 180,E1 -14424.825,E2 -14424.825} C_VEL
LIN {X 0,Y 334.775,Z 459.017,A -85,B 0,C 180,E1 -14428.152,E2 -14428.152} C_VEL
LIN {X 0,Y 334.881,Z 459.465,A -85,B 0,C 180,E1 -14431.645,E2 -14431.645} C_VEL
LIN {X 0,Y 335.034,Z 460.453,A -85,B 0,C 180,E1 -14435.106,E2 -14435.106} C_VEL
LIN {X 0,Y 335.389,Z 462.194,A -85,B 0,C 180,E1 -14438.95,E2 -14438.95} C_VEL
LIN {X 0,Y 335.755,Z 464.191,A -85,B 0,C 180,E1 -14442.053,E2 -14442.053} C_VEL
LIN {X 0,Y 336.173,Z 466.811,A -85,B 0,C 180,E1 -14445.3,E2 -14445.3} C_VEL
LIN {X 0,Y 336.555,Z 469.492,A -85,B 0,C 180,E1 -14448.07,E2 -14448.07} C_VEL
LIN {X 0,Y 336.638,Z 472.325,A -85,B 0,C 180,E1 -14450.574,E2 -14450.574} C_VEL
LIN {X 0,Y 336.286,Z 475.04,A -85,B 0,C 180,E1 -14452.695,E2 -14452.695} C_VEL
LIN {X 0,Y 335.335,Z 480.1,A -85,B 0,C 180,E1 -14456.263,E2 -14456.263} C_VEL
LIN {X 0,Y 334.498,Z 485.459,A -85,B 0,C 180,E1 -14459.719,E2 -14459.719} C_VEL
LIN {X 0,Y 334.295,Z 487.239,A -85,B 0,C 180,E1 -14460.681,E2 -14460.681} C_VEL
LIN {X 0,Y 335.358,Z 490.743,A -85,B 0,C 180,E1 -14461.009,E2 -14461.009} C_VEL
LIN {X 0,Y 336.15,Z 492.879,A -85,B 0,C 180,E1 -14461.231,E2 -14461.231} C_VEL
LIN {X 0,Y 339.855,Z 504.849,A -85,B 0,C 180,E1 -14462.412,E2 -14462.412} C_VEL
LIN {X 0,Y 342.824,Z 518.624,A -85,B 0,C 180,E1 -14463.759,E2 -14463.759} C_VEL
LIN {X 0,Y 344.199,Z 530.331,A -85,B 0,C 180,E1 -14464.91,E2 -14464.91} C_VEL
LIN {X 0,Y 344.48,Z 543.035,A -85,B 0,C 180,E1 -14466.239,E2 -14466.239} C_VEL
LIN {X 0,Y 342.886,Z 552.994,A -85,B 0,C 180,E1 -14467.271,E2 -14467.271} C_VEL
LIN {X 0,Y 340.654,Z 565.542,A -85,B 0,C 180,E1 -14468.836,E2 -14468.836} C_VEL
LIN {X 0,Y 338.438,Z 577.111,A -85,B 0,C 180,E1 -14470.595,E2 -14470.595} C_VEL
LIN {X 0,Y 336.655,Z 586.786,A -85,B 0,C 180,E1 -14472.38,E2 -14472.38} C_VEL
LIN {X 0,Y 334.979,Z 596.203,A -85,B 0,C 180,E1 -14474.47,E2 -14474.47} C_VEL
LIN {X 0,Y 333.764,Z 604.014,A -85,B 0,C 180,E1 -14476.608,E2 -14476.608} C_VEL
LIN {X 0,Y 333.004,Z 609.456,A -85,B 0,C 180,E1 -14478.434,E2 -14478.434} C_VEL
LIN {X 0,Y 332.367,Z 615.302,A -85,B 0,C 180,E1 -14480.875,E2 -14480.875} C_VEL
LIN {X 0,Y 332.167,Z 618.615,A -85,B 0,C 180,E1 -14482.707,E2 -14482.707} C_VEL
LIN {X 0,Y 332.053,Z 621.785,A -85,B 0,C 180,E1 -14485.144,E2 -14485.144} C_VEL
LIN {X 0,Y 332.092,Z 623.538,A -85,B 0,C 180,E1 -14487.574,E2 -14487.574} C_VEL
LIN {X 0,Y 332.236,Z 623.896,A -85,B 0,C 180,E1 -14488.788,E2 -14488.788} C_VEL
LIN {X 0,Y 332.266,Z 623.537,A -85,B 0,C 180,E1 -14491.212,E2 -14491.212} C_VEL
LIN {X 0,Y 332.08,Z 621.722,A -85,B 0,C 180,E1 -14493.64,E2 -14493.64} C_VEL
LIN {X 0,Y 332.128,Z 620.26,A -85,B 0,C 180,E1 -14494.855,E2 -14494.855} C_VEL
LIN {X 0,Y 332.175,Z 617.338,A -85,B 0,C 180,E1 -14496.682,E2 -14496.682} C_VEL
LIN {X 0,Y 332.311,Z 613.511,A -85,B 0,C 180,E1 -14498.513,E2 -14498.513} C_VEL
LIN {X 0,Y 332.608,Z 608.738,A -85,B 0,C 180,E1 -14500.347,E2 -14500.347} C_VEL
LIN {X 0,Y 333.269,Z 601.784,A -85,B 0,C 180,E1 -14502.483,E2 -14502.483} C_VEL
LIN {X 0,Y 333.954,Z 594.285,A -85,B 0,C 180,E1 -14504.362,E2 -14504.362} C_VEL
LIN {X 0,Y 335.074,Z 585.747,A -85,B 0,C 180,E1 -14506.135,E2 -14506.135} C_VEL
LIN {X 0,Y 336.371,Z 575.178,A -85,B 0,C 180,E1 -14507.949,E2 -14507.949} C_VEL
LIN {X 0,Y 338,Z 563.473,A -85,B 0,C 180,E1 -14509.59,E2 -14509.59} C_VEL
LIN {X 0,Y 339.376,Z 552.377,A -85,B 0,C 180,E1 -14510.869,E2 -14510.869} C_VEL
LIN {X 0,Y 340.639,Z 540.936,A -85,B 0,C 180,E1 -14511.959,E2 -14511.959} C_VEL
LIN {X 0,Y 339.296,Z 527.826,A -85,B 0,C 180,E1 -14513.095,E2 -14513.095} C_VEL
LIN {X 0,Y 337.002,Z 513.012,A -85,B 0,C 180,E1 -14514.164,E2 -14514.164} C_VEL
LIN {X 0,Y 334.386,Z 498.274,A -85,B 0,C 180,E1 -14514.989,E2 -14514.989} C_VEL
LIN {X 0,Y 333.462,Z 492.918,A -85,B 0,C 180,E1 -14515.25,E2 -14515.25} C_VEL
LIN {X 0,Y 334.107,Z 486.323,A -85,B 0,C 180,E1 -14518.934,E2 -14518.934} C_VEL
LIN {X 0,Y 334.774,Z 480.427,A -85,B 0,C 180,E1 -14522.296,E2 -14522.296} C_VEL
LIN {X 0,Y 335.619,Z 474.27,A -85,B 0,C 180,E1 -14525.896,E2 -14525.896} C_VEL
LIN {X 0,Y 336.281,Z 468.562,A -85,B 0,C 180,E1 -14529.352,E2 -14529.352} C_VEL
LIN {X 0,Y 335.812,Z 464.415,A -85,B 0,C 180,E1 -14532.044,E2 -14532.044} C_VEL
LIN {X 0,Y 334.907,Z 459.328,A -85,B 0,C 180,E1 -14535.518,E2 -14535.518} C_VEL
LIN {X 0,Y 333.983,Z 454.128,A -85,B 0,C 180,E1 -14539.282,E2 -14539.282} C_VEL
LIN {X 0,Y 333.687,Z 452.546,A -85,B 0,C 180,E1 -14540.619,E2 -14540.619} C_VEL
LIN {X 0,Y 333.672,Z 452.544,A -85,B 0,C 180,E1 -14543.861,E2 -14543.861} C_VEL
LIN {X 0,Y 333.647,Z 452.549,A -85,B 0,C 180,E1 -14547.411,E2 -14547.411} C_VEL
LIN {X 0,Y 333.707,Z 452.545,A -85,B 0,C 180,E1 -14551.028,E2 -14551.028} C_VEL
LIN {X 0,Y 333.731,Z 452.536,A -85,B 0,C 180,E1 -14553.754,E2 -14553.754} C_VEL
LIN {X 0,Y 333.715,Z 452.538,A -85,B 0,C 180,E1 -14557.914,E2 -14557.914} C_VEL
LIN {X 0,Y 333.788,Z 452.529,A -85,B 0,C 180,E1 -14561.589,E2 -14561.589} C_VEL
LIN {X 0,Y 333.803,Z 452.527,A -85,B 0,C 180,E1 -14565.577,E2 -14565.577} C_VEL
LIN {X 0,Y 333.828,Z 452.527,A -85,B 0,C 180,E1 -14569.078,E2 -14569.078} C_VEL
LIN {X 0,Y 334.02,Z 452.506,A -85,B 0,C 180,E1 -14572.748,E2 -14572.748} C_VEL
LIN {X 0,Y 333.807,Z 452.528,A -85,B 0,C 180,E1 -14575.169,E2 -14575.169} C_VEL
LIN {X 0,Y 334.102,Z 452.49,A -85,B 0,C 180,E1 -14577.589,E2 -14577.589} C_VEL
LIN {X 0,Y 334.241,Z 452.473,A -85,B 0,C 180,E1 -14580,E2 -14580} C_VEL
LIN {X 0,Y 334.127,Z 452.491,A -85,B 0,C 180,E1 -14582.411,E2 -14582.411} C_VEL
LIN {X 0,Y 334.023,Z 452.5,A -85,B 0,C 180,E1 -14587.253,E2 -14587.253} C_VEL
LIN {X 0,Y 333.828,Z 452.526,A -85,B 0,C 180,E1 -14590.922,E2 -14590.922} C_VEL
LIN {X 0,Y 333.804,Z 452.531,A -85,B 0,C 180,E1 -14594.635,E2 -14594.635} C_VEL
LIN {X 0,Y 333.793,Z 452.531,A -85,B 0,C 180,E1 -14598.656,E2 -14598.656} C_VEL
LIN {X 0,Y 333.688,Z 452.547,A -85,B 0,C 180,E1 -14602.279,E2 -14602.279} C_VEL
LIN {X 0,Y 333.732,Z 452.542,A -85,B 0,C 180,E1 -14606.247,E2 -14606.247} C_VEL
LIN {X 0,Y 333.707,Z 452.539,A -85,B 0,C 180,E1 -14608.973,E2 -14608.973} C_VEL
LIN {X 0,Y 333.64,Z 452.549,A -85,B 0,C 180,E1 -14612.588,E2 -14612.588} C_VEL
LIN {X 0,Y 333.674,Z 452.549,A -85,B 0,C 180,E1 -14616.14,E2 -14616.14} C_VEL
LIN {X 0,Y 333.645,Z 452.547,A -85,B 0,C 180,E1 -14619.193,E2 -14619.193} C_VEL
LIN {X 0,Y 333.631,Z 452.55,A -85,B 0,C 180,E1 -14622.501,E2 -14622.501} C_VEL
LIN {X 0,Y 333.608,Z 452.557,A -85,B 0,C 180,E1 -14625.958,E2 -14625.958} C_VEL
LIN {X 0,Y 333.656,Z 452.546,A -85,B 0,C 180,E1 -14629.314,E2 -14629.314} C_VEL
LIN {X 0,Y 333.656,Z 452.547,A -85,B 0,C 180,E1 -14632.35,E2 -14632.35} C_VEL
LIN {X 0,Y 333.675,Z 452.544,A -85,B 0,C 180,E1 -14635.342,E2 -14635.342} C_VEL
LIN {X 0,Y 333.704,Z 452.544,A -85,B 0,C 180,E1 -14639.711,E2 -14639.711} C_VEL
LIN {X 0,Y 333.746,Z 452.535,A -85,B 0,C 180,E1 -14642.402,E2 -14642.402} C_VEL
LIN {X 0,Y 333.729,Z 452.537,A -85,B 0,C 180,E1 -14645.091,E2 -14645.091} C_VEL
LIN {X 0,Y 333.684,Z 452.543,A -85,B 0,C 180,E1 -14649.02,E2 -14649.02} C_VEL
LIN {X 0,Y 333.797,Z 452.533,A -85,B 0,C 180,E1 -14651.59,E2 -14651.59} C_VEL
LIN {X 0,Y 333.811,Z 452.532,A -85,B 0,C 180,E1 -14655.577,E2 -14655.577} C_VEL
LIN {X 0,Y 333.837,Z 452.525,A -85,B 0,C 180,E1 -14659.078,E2 -14659.078} C_VEL
LIN {X 0,Y 333.972,Z 452.507,A -85,B 0,C 180,E1 -14662.746,E2 -14662.746} C_VEL
LIN {X 0,Y 333.807,Z 452.53,A -85,B 0,C 180,E1 -14665.169,E2 -14665.169} C_VEL
LIN {X 0,Y 334.11,Z 452.493,A -85,B 0,C 180,E1 -14667.589,E2 -14667.589} C_VEL
LIN {X 0,Y 334.25,Z 452.472,A -85,B 0,C 180,E1 -14670,E2 -14670} C_VEL
LIN {X 0,Y 334.109,Z 452.489,A -85,B 0,C 180,E1 -14672.411,E2 -14672.411} C_VEL
LIN {X 0,Y 334.017,Z 452.501,A -85,B 0,C 180,E1 -14676.039,E2 -14676.039} C_VEL
LIN {X 0,Y 333.962,Z 452.508,A -85,B 0,C 180,E1 -14678.471,E2 -14678.471} C_VEL
LIN {X 0,Y 333.795,Z 452.528,A -85,B 0,C 180,E1 -14682.154,E2 -14682.154} C_VEL
LIN {X 0,Y 333.781,Z 452.53,A -85,B 0,C 180,E1 -14685.886,E2 -14685.886} C_VEL
LIN {X 0,Y 333.798,Z 452.529,A -85,B 0,C 180,E1 -14688.654,E2 -14688.654} C_VEL
LIN {X 0,Y 333.695,Z 452.541,A -85,B 0,C 180,E1 -14692.278,E2 -14692.278} C_VEL
LIN {X 0,Y 333.737,Z 452.536,A -85,B 0,C 180,E1 -14696.246,E2 -14696.246} C_VEL
LIN {X 0,Y 333.712,Z 452.544,A -85,B 0,C 180,E1 -14698.971,E2 -14698.971} C_VEL
LIN {X 0,Y 333.637,Z 452.55,A -85,B 0,C 180,E1 -14702.584,E2 -14702.584} C_VEL
LIN {X 0,Y 333.564,Z 452.561,A -85,B 0,C 180,E1 -14704.743,E2 -14704.743} C_VEL
LIN {X 0,Y 333.236,Z 452.598,A -85,B 0,C 180,E1 -14707.706,E2 -14707.706} C_VEL
LIN {X 0,Y 332.839,Z 452.653,A -85,B 0,C 180,E1 -14710.886,E2 -14710.886} C_VEL
LIN {X 0,Y 332.671,Z 452.879,A -85,B 0,C 180,E1 -14712.533,E2 -14712.533} C_VEL
LIN {X 0,Y 332.556,Z 455.647,A -85,B 0,C 180,E1 -14715.932,E2 -14715.932} C_VEL
LIN {X 0,Y 332.555,Z 456.507,A -85,B 0,C 180,E1 -14716.913,E2 -14716.913} C_VEL
LIN {X 0,Y 336.776,Z 471.185,A -85,B 0,C 180,E1 -14717.801,E2 -14717.801} C_VEL
LIN {X 0,Y 340.326,Z 484.853,A -85,B 0,C 180,E1 -14718.825,E2 -14718.825} C_VEL
LIN {X 0,Y 342.257,Z 493.247,A -85,B 0,C 180,E1 -14719.556,E2 -14719.556} C_VEL
LIN {X 0,Y 341.042,Z 506.505,A -85,B 0,C 180,E1 -14720.677,E2 -14720.677} C_VEL
LIN {X 0,Y 339.591,Z 519.094,A -85,B 0,C 180,E1 -14721.997,E2 -14721.997} C_VEL
LIN {X 0,Y 338.219,Z 530.768,A -85,B 0,C 180,E1 -14723.501,E2 -14723.501} C_VEL
LIN {X 0,Y 337.003,Z 540.48,A -85,B 0,C 180,E1 -14725.005,E2 -14725.005} C_VEL
LIN {X 0,Y 335.762,Z 550.437,A -85,B 0,C 180,E1 -14726.856,E2 -14726.856} C_VEL
LIN {X 0,Y 334.581,Z 554.176,A -85,B 0,C 180,E1 -14727.612,E2 -14727.612} C_VEL
LIN {X 0,Y 331.029,Z 559.906,A -85,B 0,C 180,E1 -14728.865,E2 -14728.865} C_VEL
LIN {X 0,Y 327.581,Z 565.084,A -85,B 0,C 180,E1 -14730.209,E2 -14730.209} C_VEL
LIN {X 0,Y 326.579,Z 567.957,A -85,B 0,C 180,E1 -14731.097,E2 -14731.097} C_VEL
LIN {X 0,Y 325.933,Z 573.451,A -85,B 0,C 180,E1 -14733.075,E2 -14733.075} C_VEL
LIN {X 0,Y 325.516,Z 577.872,A -85,B 0,C 180,E1 -14735.064,E2 -14735.064} C_VEL
LIN {X 0,Y 325.156,Z 581.32,A -85,B 0,C 180,E1 -14737.104,E2 -14737.104} C_VEL
LIN {X 0,Y 325.042,Z 583.055,A -85,B 0,C 180,E1 -14738.434,E2 -14738.434} C_VEL
LIN {X 0,Y 324.928,Z 584.352,A -85,B 0,C 180,E1 -14739.752,E2 -14739.752} C_VEL
LIN {X 0,Y 324.958,Z 585.763,A -85,B 0,C 180,E1 -14742.375,E2 -14742.375} C_VEL
LIN {X 0,Y 325.091,Z 585.692,A -85,B 0,C 180,E1 -14744.964,E2 -14744.964} C_VEL
LIN {X 0,Y 325.511,Z 584.184,A -85,B 0,C 180,E1 -14747.531,E2 -14747.531} C_VEL
LIN {X 0,Y 326.153,Z 581.263,A -85,B 0,C 180,E1 -14750.073,E2 -14750.073} C_VEL
LIN {X 0,Y 326.737,Z 578.637,A -85,B 0,C 180,E1 -14751.66,E2 -14751.66} C_VEL
LIN {X 0,Y 327.725,Z 574.011,A -85,B 0,C 180,E1 -14753.844,E2 -14753.844} C_VEL
LIN {X 0,Y 329.307,Z 567.121,A -85,B 0,C 180,E1 -14756.329,E2 -14756.329} C_VEL
LIN {X 0,Y 330.843,Z 560.329,A -85,B 0,C 180,E1 -14758.279,E2 -14758.279} C_VEL
LIN {X 0,Y 332.762,Z 551.697,A -85,B 0,C 180,E1 -14760.302,E2 -14760.302} C_VEL
LIN {X 0,Y 334.824,Z 542.303,A -85,B 0,C 180,E1 -14762.105,E2 -14762.105} C_VEL
LIN {X 0,Y 337.161,Z 531.058,A -85,B 0,C 180,E1 -14763.884,E2 -14763.884} C_VEL
LIN {X 0,Y 339.317,Z 519.864,A -85,B 0,C 180,E1 -14765.325,E2 -14765.325} C_VEL
LIN {X 0,Y 341.4,Z 507.525,A -85,B 0,C 180,E1 -14766.625,E2 -14766.625} C_VEL
LIN {X 0,Y 342.148,Z 502.564,A -85,B 0,C 180,E1 -14767.079,E2 -14767.079} C_VEL
LIN {X 0,Y 339.701,Z 491.691,A -85,B 0,C 180,E1 -14768.464,E2 -14768.464} C_VEL
LIN {X 0,Y 335.404,Z 480.342,A -85,B 0,C 180,E1 -14769.998,E2 -14769.998} C_VEL
LIN {X 0,Y 330.749,Z 471.064,A -85,B 0,C 180,E1 -14771.345,E2 -14771.345} C_VEL
LIN {X 0,Y 328.922,Z 467.599,A -85,B 0,C 180,E1 -14771.868,E2 -14771.868} C_VEL
LIN {X 0,Y 327.396,Z 464.973,A -85,B 0,C 180,E1 -14772.278,E2 -14772.278} C_VEL
LIN {X 0,Y 327.075,Z 463.713,A -85,B 0,C 180,E1 -14772.408,E2 -14772.408} C_VEL
LIN {X 0,Y 327.378,Z 462.298,A -85,B 0,C 180,E1 -14776.205,E2 -14776.205} C_VEL
LIN {X 0,Y 327.69,Z 461.375,A -85,B 0,C 180,E1 -14779.325,E2 -14779.325} C_VEL
LIN {X 0,Y 327.749,Z 460.719,A -85,B 0,C 180,E1 -14782.773,E2 -14782.773} C_VEL
LIN {X 0,Y 327.831,Z 460.474,A -85,B 0,C 180,E1 -14785.793,E2 -14785.793} C_VEL
LIN {X 0,Y 327.865,Z 460.647,A -85,B 0,C 180,E1 -14789.539,E2 -14789.539} C_VEL
LIN {X 0,Y 328.011,Z 461.403,A -85,B 0,C 180,E1 -14793.321,E2 -14793.321} C_VEL
LIN {X 0,Y 328.236,Z 462.694,A -85,B 0,C 180,E1 -14796.835,E2 -14796.835} C_VEL
LIN {X 0,Y 328.55,Z 464.31,A -85,B 0,C 180,E1 -14799.921,E2 -14799.921} C_VEL
LIN {X 0,Y 328.997,Z 466.732,A -85,B 0,C 180,E1 -14803.424,E2 -14803.424} C_VEL
LIN {X 0,Y 329.485,Z 469.808,A -85,B 0,C 180,E1 -14806.956,E2 -14806.956} C_VEL
LIN {X 0,Y 329.675,Z 473.151,A -85,B 0,C 180,E1 -14810.125,E2 -14810.125} C_VEL
LIN {X 0,Y 329.381,Z 475.615,A -85,B 0,C 180,E1 -14812.136,E2 -14812.136} C_VEL
LIN {X 0,Y 328.526,Z 480.13,A -85,B 0,C 180,E1 -14815.466,E2 -14815.466} C_VEL
LIN {X 0,Y 327.591,Z 485.555,A -85,B 0,C 180,E1 -14819.109,E2 -14819.109} C_VEL
LIN {X 0,Y 327.491,Z 486.301,A -85,B 0,C 180,E1 -14819.592,E2 -14819.592} C_VEL
LIN {X 0,Y 328.435,Z 489.804,A -85,B 0,C 180,E1 -14819.94,E2 -14819.94} C_VEL
LIN {X 0,Y 329.519,Z 492.523,A -85,B 0,C 180,E1 -14820.248,E2 -14820.248} C_VEL
LIN {X 0,Y 332.99,Z 503.215,A -85,B 0,C 180,E1 -14821.408,E2 -14821.408} C_VEL
LIN {X 0,Y 335.938,Z 515.818,A -85,B 0,C 180,E1 -14822.717,E2 -14822.717} C_VEL
LIN {X 0,Y 337.552,Z 526.729,A -85,B 0,C 180,E1 -14823.859,E2 -14823.859} C_VEL
LIN {X 0,Y 338.162,Z 539.065,A -85,B 0,C 180,E1 -14825.174,E2 -14825.174} C_VEL
LIN {X 0,Y 337.78,Z 547.085,A -85,B 0,C 180,E1 -14826.064,E2 -14826.064} C_VEL
LIN {X 0,Y 335.647,Z 557.875,A -85,B 0,C 180,E1 -14827.286,E2 -14827.286} C_VEL
LIN {X 0,Y 333.245,Z 570.141,A -85,B 0,C 180,E1 -14828.991,E2 -14828.991} C_VEL
LIN {X 0,Y 331.082,Z 580.853,A -85,B 0,C 180,E1 -14830.791,E2 -14830.791} C_VEL
LIN {X 0,Y 329.059,Z 591.234,A -85,B 0,C 180,E1 -14832.922,E2 -14832.922} C_VEL
LIN {X 0,Y 327.493,Z 599.772,A -85,B 0,C 180,E1 -14835.077,E2 -14835.077} C_VEL
LIN {X 0,Y 326.538,Z 605.846,A -85,B 0,C 180,E1 -14836.939,E2 -14836.939} C_VEL
LIN {X 0,Y 325.577,Z 612.432,A -85,B 0,C 180,E1 -14839.427,E2 -14839.427} C_VEL
LIN {X 0,Y 325.139,Z 617.361,A -85,B 0,C 180,E1 -14841.923,E2 -14841.923} C_VEL
LIN {X 0,Y 324.974,Z 620.541,A -85,B 0,C 180,E1 -14844.16,E2 -14844.16} C_VEL
LIN {X 0,Y 324.986,Z 622.478,A -85,B 0,C 180,E1 -14846.28,E2 -14846.28} C_VEL
LIN {X 0,Y 325.14,Z 623.477,A -85,B 0,C 180,E1 -14848.761,E2 -14848.761} C_VEL
LIN {X 0,Y 325.21,Z 623.445,A -85,B 0,C 180,E1 -14850,E2 -14850} C_VEL
LIN {X 0,Y 325.186,Z 623.047,A -85,B 0,C 180,E1 -14851.238,E2 -14851.238} C_VEL
LIN {X 0,Y 325.007,Z 621.149,A -85,B 0,C 180,E1 -14853.719,E2 -14853.719} C_VEL
LIN {X 0,Y 325.106,Z 617.777,A -85,B 0,C 180,E1 -14856.205,E2 -14856.205} C_VEL
LIN {X 0,Y 325.191,Z 614.239,A -85,B 0,C 180,E1 -14858.075,E2 -14858.075} C_VEL
LIN {X 0,Y 325.431,Z 609.691,A -85,B 0,C 180,E1 -14859.949,E2 -14859.949} C_VEL
LIN {X 0,Y 326.069,Z 603.115,A -85,B 0,C 180,E1 -14862.131,E2 -14862.131} C_VEL
LIN {X 0,Y 326.748,Z 595.795,A -85,B 0,C 180,E1 -14864.095,E2 -14864.095} C_VEL
LIN {X 0,Y 327.954,Z 586.331,A -85,B 0,C 180,E1 -14866.176,E2 -14866.176} C_VEL
LIN {X 0,Y 329.303,Z 575.973,A -85,B 0,C 180,E1 -14868.026,E2 -14868.026} C_VEL
LIN {X 0,Y 330.909,Z 564.503,A -85,B 0,C 180,E1 -14869.704,E2 -14869.704} C_VEL
LIN {X 0,Y 332.395,Z 553.182,A -85,B 0,C 180,E1 -14871.065,E2 -14871.065} C_VEL
LIN {X 0,Y 333.706,Z 540.945,A -85,B 0,C 180,E1 -14872.277,E2 -14872.277} C_VEL
LIN {X 0,Y 332.229,Z 527.632,A -85,B 0,C 180,E1 -14873.465,E2 -14873.465} C_VEL
LIN {X 0,Y 330.138,Z 513.831,A -85,B 0,C 180,E1 -14874.486,E2 -14874.486} C_VEL
LIN {X 0,Y 327.547,Z 498.741,A -85,B 0,C 180,E1 -14875.368,E2 -14875.368} C_VEL
LIN {X 0,Y 326.437,Z 492.567,A -85,B 0,C 180,E1 -14875.685,E2 -14875.685} C_VEL
LIN {X 0,Y 327.146,Z 485.735,A -85,B 0,C 180,E1 -14879.61,E2 -14879.61} C_VEL
LIN {X 0,Y 327.931,Z 479.46,A -85,B 0,C 180,E1 -14883.299,E2 -14883.299} C_VEL
LIN {X 0,Y 328.715,Z 473.694,A -85,B 0,C 180,E1 -14886.772,E2 -14886.772} C_VEL
LIN {X 0,Y 329.172,Z 470.083,A -85,B 0,C 180,E1 -14889.014,E2 -14889.014} C_VEL
LIN {X 0,Y 328.91,Z 466.14,A -85,B 0,C 180,E1 -14891.594,E2 -14891.594} C_VEL
LIN {X 0,Y 328.049,Z 461.211,A -85,B 0,C 180,E1 -14895.01,E2 -14895.01} C_VEL
LIN {X 0,Y 327.128,Z 456.089,A -85,B 0,C 180,E1 -14898.757,E2 -14898.757} C_VEL
LIN {X 0,Y 326.664,Z 453.421,A -85,B 0,C 180,E1 -14900.869,E2 -14900.869} C_VEL
LIN {X 0,Y 326.615,Z 453.426,A -85,B 0,C 180,E1 -14904.851,E2 -14904.851} C_VEL
LIN {X 0,Y 326.611,Z 453.425,A -85,B 0,C 180,E1 -14907.456,E2 -14907.456} C_VEL
LIN {X 0,Y 326.657,Z 453.418,A -85,B 0,C 180,E1 -14910.341,E2 -14910.341} C_VEL
LIN {X 0,Y 326.685,Z 453.415,A -85,B 0,C 180,E1 -14914.516,E2 -14914.516} C_VEL
LIN {X 0,Y 326.643,Z 453.421,A -85,B 0,C 180,E1 -14918.545,E2 -14918.545} C_VEL
LIN {X 0,Y 326.74,Z 453.41,A -85,B 0,C 180,E1 -14921.177,E2 -14921.177} C_VEL
LIN {X 0,Y 326.758,Z 453.405,A -85,B 0,C 180,E1 -14925.433,E2 -14925.433} C_VEL
LIN {X 0,Y 326.764,Z 453.409,A -85,B 0,C 180,E1 -14928.839,E2 -14928.839} C_VEL
LIN {X 0,Y 326.974,Z 453.382,A -85,B 0,C 180,E1 -14932.59,E2 -14932.59} C_VEL
LIN {X 0,Y 326.774,Z 453.405,A -85,B 0,C 180,E1 -14935.065,E2 -14935.065} C_VEL
LIN {X 0,Y 327.043,Z 453.369,A -85,B 0,C 180,E1 -14937.537,E2 -14937.537} C_VEL
LIN {X 0,Y 327.193,Z 453.351,A -85,B 0,C 180,E1 -14940,E2 -14940} C_VEL
LIN {X 0,Y 327.064,Z 453.371,A -85,B 0,C 180,E1 -14942.463,E2 -14942.463} C_VEL
LIN {X 0,Y 326.971,Z 453.377,A -85,B 0,C 180,E1 -14946.598,E2 -14946.598} C_VEL
LIN {X 0,Y 326.809,Z 453.399,A -85,B 0,C 180,E1 -14949.907,E2 -14949.907} C_VEL
LIN {X 0,Y 326.754,Z 453.405,A -85,B 0,C 180,E1 -14953.686,E2 -14953.686} C_VEL
LIN {X 0,Y 326.694,Z 453.413,A -85,B 0,C 180,E1 -14957.528,E2 -14957.528} C_VEL
LIN {X 0,Y 326.661,Z 453.421,A -85,B 0,C 180,E1 -14960.135,E2 -14960.135} C_VEL
LIN {X 0,Y 326.648,Z 453.423,A -85,B 0,C 180,E1 -14964.13,E2 -14964.13} C_VEL
LIN {X 0,Y 326.68,Z 453.415,A -85,B 0,C 180,E1 -14966.858,E2 -14966.858} C_VEL
LIN {X 0,Y 326.636,Z 453.422,A -85,B 0,C 180,E1 -14970.612,E2 -14970.612} C_VEL
LIN {X 0,Y 326.604,Z 453.428,A -85,B 0,C 180,E1 -14974.02,E2 -14974.02} C_VEL
LIN {X 0,Y 326.625,Z 453.421,A -85,B 0,C 180,E1 -14977.239,E2 -14977.239} C_VEL
LIN {X 0,Y 326.576,Z 453.427,A -85,B 0,C 180,E1 -14981.132,E2 -14981.132} C_VEL
LIN {X 0,Y 326.53,Z 453.433,A -85,B 0,C 180,E1 -14984.744,E2 -14984.744} C_VEL
LIN {X 0,Y 326.597,Z 453.428,A -85,B 0,C 180,E1 -14988.158,E2 -14988.158} C_VEL
LIN {X 0,Y 326.643,Z 453.42,A -85,B 0,C 180,E1 -14991.395,E2 -14991.395} C_VEL
LIN {X 0,Y 326.62,Z 453.422,A -85,B 0,C 180,E1 -14994.852,E2 -14994.852} C_VEL
LIN {X 0,Y 326.611,Z 453.425,A -85,B 0,C 180,E1 -14997.457,E2 -14997.457} C_VEL
LIN {X 0,Y 326.662,Z 453.418,A -85,B 0,C 180,E1 -15000.342,E2 -15000.342} C_VEL
LIN {X 0,Y 326.687,Z 453.414,A -85,B 0,C 180,E1 -15003.143,E2 -15003.143} C_VEL
LIN {X 0,Y 326.654,Z 453.422,A -85,B 0,C 180,E1 -15005.872,E2 -15005.872} C_VEL
LIN {X 0,Y 326.668,Z 453.42,A -85,B 0,C 180,E1 -15009.866,E2 -15009.866} C_VEL
LIN {X 0,Y 326.702,Z 453.412,A -85,B 0,C 180,E1 -15012.473,E2 -15012.473} C_VEL
LIN {X 0,Y 326.762,Z 453.404,A -85,B 0,C 180,E1 -15016.315,E2 -15016.315} C_VEL
LIN {X 0,Y 326.808,Z 453.399,A -85,B 0,C 180,E1 -15020.094,E2 -15020.094} C_VEL
LIN {X 0,Y 326.956,Z 453.382,A -85,B 0,C 180,E1 -15023.83,E2 -15023.83} C_VEL
LIN {X 0,Y 327.051,Z 453.373,A -85,B 0,C 180,E1 -15027.537,E2 -15027.537} C_VEL
LIN {X 0,Y 327.201,Z 453.35,A -85,B 0,C 180,E1 -15030,E2 -15030} C_VEL
LIN {X 0,Y 327.05,Z 453.368,A -85,B 0,C 180,E1 -15032.463,E2 -15032.463} C_VEL
LIN {X 0,Y 326.991,Z 453.376,A -85,B 0,C 180,E1 -15036.169,E2 -15036.169} C_VEL
LIN {X 0,Y 326.809,Z 453.399,A -85,B 0,C 180,E1 -15039.906,E2 -15039.906} C_VEL
LIN {X 0,Y 326.762,Z 453.406,A -85,B 0,C 180,E1 -15043.685,E2 -15043.685} C_VEL
LIN {X 0,Y 326.702,Z 453.414,A -85,B 0,C 180,E1 -15047.527,E2 -15047.527} C_VEL
LIN {X 0,Y 326.668,Z 453.416,A -85,B 0,C 180,E1 -15050.134,E2 -15050.134} C_VEL
LIN {X 0,Y 326.654,Z 453.417,A -85,B 0,C 180,E1 -15054.128,E2 -15054.128} C_VEL
LIN {X 0,Y 326.686,Z 453.418,A -85,B 0,C 180,E1 -15056.857,E2 -15056.857} C_VEL
LIN {X 0,Y 326.639,Z 453.422,A -85,B 0,C 180,E1 -15060.61,E2 -15060.61} C_VEL
LIN {X 0,Y 326.55,Z 453.43,A -85,B 0,C 180,E1 -15064.025,E2 -15064.025} C_VEL
LIN {X 0,Y 326.257,Z 453.47,A -85,B 0,C 180,E1 -15067.152,E2 -15067.152} C_VEL
LIN {X 0,Y 325.802,Z 453.529,A -85,B 0,C 180,E1 -15070.974,E2 -15070.974} C_VEL
LIN {X 0,Y 325.598,Z 453.846,A -85,B 0,C 180,E1 -15072.786,E2 -15072.786} C_VEL
LIN {X 0,Y 325.511,Z 457.024,A -85,B 0,C 180,E1 -15076.483,E2 -15076.483} C_VEL
LIN {X 0,Y 329.921,Z 472.317,A -85,B 0,C 180,E1 -15077.448,E2 -15077.448} C_VEL
LIN {X 0,Y 333.619,Z 486.578,A -85,B 0,C 180,E1 -15078.56,E2 -15078.56} C_VEL
LIN {X 0,Y 335.347,Z 494.229,A -85,B 0,C 180,E1 -15079.25,E2 -15079.25} C_VEL
LIN {X 0,Y 334.27,Z 506.447,A -85,B 0,C 180,E1 -15080.31,E2 -15080.31} C_VEL
LIN {X 0,Y 332.69,Z 519.839,A -85,B 0,C 180,E1 -15081.744,E2 -15081.744} C_VEL
LIN {X 0,Y 331.205,Z 532.009,A -85,B 0,C 180,E1 -15083.359,E2 -15083.359} C_VEL
LIN {X 0,Y 329.949,Z 541.574,A -85,B 0,C 180,E1 -15084.892,E2 -15084.892} C_VEL
LIN {X 0,Y 328.743,Z 550.964,A -85,B 0,C 180,E1 -15086.689,E2 -15086.689} C_VEL
LIN {X 0,Y 327.542,Z 559.458,A -85,B 0,C 180,E1 -15088.645,E2 -15088.645} C_VEL
LIN {X 0,Y 326.689,Z 566.739,A -85,B 0,C 180,E1 -15090.697,E2 -15090.697} C_VEL
LIN {X 0,Y 326.579,Z 567.957,A -85,B 0,C 180,E1 -15091.097,E2 -15091.097} C_VEL
LIN {X 0,Y 325.603,Z 570.687,A -85,B 0,C 180,E1 -15092.005,E2 -15092.005} C_VEL
LIN {X 0,Y 322.316,Z 574.75,A -85,B 0,C 180,E1 -15093.494,E2 -15093.494} C_VEL
LIN {X 0,Y 319.089,Z 578.27,A -85,B 0,C 180,E1 -15095.053,E2 -15095.053} C_VEL
LIN {X 0,Y 318.231,Z 580.077,A -85,B 0,C 180,E1 -15096.057,E2 -15096.057} C_VEL
LIN {X 0,Y 317.945,Z 583.116,A -85,B 0,C 180,E1 -15098.182,E2 -15098.182} C_VEL
LIN {X 0,Y 317.802,Z 585.358,A -85,B 0,C 180,E1 -15100.627,E2 -15100.627} C_VEL
LIN {X 0,Y 317.851,Z 586.056,A -85,B 0,C 180,E1 -15101.967,E2 -15101.967} C_VEL
LIN {X 0,Y 317.979,Z 586.313,A -85,B 0,C 180,E1 -15104.619,E2 -15104.619} C_VEL
LIN {X 0,Y 318.387,Z 585.088,A -85,B 0,C 180,E1 -15107.247,E2 -15107.247} C_VEL
LIN {X 0,Y 319.013,Z 582.45,A -85,B 0,C 180,E1 -15109.849,E2 -15109.849} C_VEL
LIN {X 0,Y 320.006,Z 578.362,A -85,B 0,C 180,E1 -15112.428,E2 -15112.428} C_VEL
LIN {X 0,Y 321.365,Z 572.752,A -85,B 0,C 180,E1 -15114.981,E2 -15114.981} C_VEL
LIN {X 0,Y 322.937,Z 566.399,A -85,B 0,C 180,E1 -15117.193,E2 -15117.193} C_VEL
LIN {X 0,Y 324.767,Z 558.545,A -85,B 0,C 180,E1 -15119.38,E2 -15119.38} C_VEL
LIN {X 0,Y 326.768,Z 550.431,A -85,B 0,C 180,E1 -15121.232,E2 -15121.232} C_VEL
LIN {X 0,Y 329.034,Z 540.714,A -85,B 0,C 180,E1 -15123.061,E2 -15123.061} C_VEL
LIN {X 0,Y 331.54,Z 528.986,A -85,B 0,C 180,E1 -15124.864,E2 -15124.864} C_VEL
LIN {X 0,Y 334.018,Z 516.413,A -85,B 0,C 180,E1 -15126.438,E2 -15126.438} C_VEL
LIN {X 0,Y 336.068,Z 504.913,A -85,B 0,C 180,E1 -15127.602,E2 -15127.602} C_VEL
LIN {X 0,Y 334.239,Z 495.899,A -85,B 0,C 180,E1 -15128.794,E2 -15128.794} C_VEL
LIN {X 0,Y 330.616,Z 485.317,A -85,B 0,C 180,E1 -15130.308,E2 -15130.308} C_VEL
LIN {X 0,Y 324.553,Z 472.714,A -85,B 0,C 180,E1 -15132.276,E2 -15132.276} C_VEL
LIN {X 0,Y 322.72,Z 469.228,A -85,B 0,C 180,E1 -15132.842,E2 -15132.842} C_VEL
LIN {X 0,Y 320.683,Z 466.25,A -85,B 0,C 180,E1 -15133.404,E2 -15133.404} C_VEL
LIN {X 0,Y 320.204,Z 464.5,A -85,B 0,C 180,E1 -15133.647,E2 -15133.647} C_VEL
LIN {X 0,Y 320.434,Z 463.51,A -85,B 0,C 180,E1 -15136.566,E2 -15136.566} C_VEL
LIN {X 0,Y 320.741,Z 462.683,A -85,B 0,C 180,E1 -15139.578,E2 -15139.578} C_VEL
LIN {X 0,Y 320.793,Z 462.112,A -85,B 0,C 180,E1 -15143.225,E2 -15143.225} C_VEL
LIN {X 0,Y 320.884,Z 461.94,A -85,B 0,C 180,E1 -15146.108,E2 -15146.108} C_VEL
LIN {X 0,Y 320.946,Z 462.272,A -85,B 0,C 180,E1 -15150.241,E2 -15150.241} C_VEL
LIN {X 0,Y 321.101,Z 463.072,A -85,B 0,C 180,E1 -15153.726,E2 -15153.726} C_VEL
LIN {X 0,Y 321.407,Z 464.681,A -85,B 0,C 180,E1 -15157.753,E2 -15157.753} C_VEL
LIN {X 0,Y 321.732,Z 466.479,A -85,B 0,C 180,E1 -15160.944,E2 -15160.944} C_VEL
LIN {X 0,Y 322.152,Z 468.912,A -85,B 0,C 180,E1 -15164.275,E2 -15164.275} C_VEL
LIN {X 0,Y 322.603,Z 472.059,A -85,B 0,C 180,E1 -15167.791,E2 -15167.791} C_VEL
LIN {X 0,Y 322.59,Z 475.327,A -85,B 0,C 180,E1 -15170.818,E2 -15170.818} C_VEL
LIN {X 0,Y 321.94,Z 479.186,A -85,B 0,C 180,E1 -15173.885,E2 -15173.885} C_VEL
LIN {X 0,Y 320.994,Z 484.315,A -85,B 0,C 180,E1 -15177.561,E2 -15177.561} C_VEL
LIN {X 0,Y 320.721,Z 485.585,A -85,B 0,C 180,E1 -15178.423,E2 -15178.423} C_VEL
LIN {X 0,Y 321.674,Z 489.029,A -85,B 0,C 180,E1 -15178.782,E2 -15178.782} C_VEL
LIN {X 0,Y 322.761,Z 491.504,A -85,B 0,C 180,E1 -15179.109,E2 -15179.109} C_VEL
LIN {X 0,Y 326.327,Z 502.262,A -85,B 0,C 180,E1 -15180.385,E2 -15180.385} C_VEL
LIN {X 0,Y 329.51,Z 515.235,A -85,B 0,C 180,E1 -15181.845,E2 -15181.845} C_VEL
LIN {X 0,Y 331.289,Z 526.609,A -85,B 0,C 180,E1 -15183.107,E2 -15183.107} C_VEL
LIN {X 0,Y 331.882,Z 539.178,A -85,B 0,C 180,E1 -15184.517,E2 -15184.517} C_VEL
LIN {X 0,Y 331.623,Z 546.846,A -85,B 0,C 180,E1 -15185.424,E2 -15185.424} C_VEL
LIN {X 0,Y 329.138,Z 558.836,A -85,B 0,C 180,E1 -15186.829,E2 -15186.829} C_VEL
LIN {X 0,Y 326.648,Z 570.743,A -85,B 0,C 180,E1 -15188.546,E2 -15188.546} C_VEL
LIN {X 0,Y 324.389,Z 581.202,A -85,B 0,C 180,E1 -15190.378,E2 -15190.378} C_VEL
LIN {X 0,Y 322.247,Z 591.444,A -85,B 0,C 180,E1 -15192.55,E2 -15192.55} C_VEL
LIN {X 0,Y 320.592,Z 599.834,A -85,B 0,C 180,E1 -15194.748,E2 -15194.748} C_VEL
LIN {X 0,Y 319.278,Z 607.551,A -85,B 0,C 180,E1 -15197.284,E2 -15197.284} C_VEL
LIN {X 0,Y 318.397,Z 613.601,A -85,B 0,C 180,E1 -15199.829,E2 -15199.829} C_VEL
LIN {X 0,Y 317.996,Z 618.095,A -85,B 0,C 180,E1 -15202.38,E2 -15202.38} C_VEL
LIN {X 0,Y 317.867,Z 621.13,A -85,B 0,C 180,E1 -15204.926,E2 -15204.926} C_VEL
LIN {X 0,Y 317.911,Z 622.121,A -85,B 0,C 180,E1 -15206.197,E2 -15206.197} C_VEL
LIN {X 0,Y 318.045,Z 623.047,A -85,B 0,C 180,E1 -15208.734,E2 -15208.734} C_VEL
LIN {X 0,Y 318.152,Z 622.977,A -85,B 0,C 180,E1 -15210,E2 -15210} C_VEL
LIN {X 0,Y 318.109,Z 622.537,A -85,B 0,C 180,E1 -15211.266,E2 -15211.266} C_VEL
LIN {X 0,Y 317.936,Z 620.566,A -85,B 0,C 180,E1 -15213.802,E2 -15213.802} C_VEL
LIN {X 0,Y 318.017,Z 617.651,A -85,B 0,C 180,E1 -15216.026,E2 -15216.026} C_VEL
LIN {X 0,Y 318.134,Z 613.511,A -85,B 0,C 180,E1 -15218.256,E2 -15218.256} C_VEL
LIN {X 0,Y 318.393,Z 608.909,A -85,B 0,C 180,E1 -15220.171,E2 -15220.171} C_VEL
LIN {X 0,Y 319.05,Z 602.238,A -85,B 0,C 180,E1 -15222.402,E2 -15222.402} C_VEL
LIN {X 0,Y 319.716,Z 595.162,A -85,B 0,C 180,E1 -15224.321,E2 -15224.321} C_VEL
LIN {X 0,Y 320.842,Z 586.744,A -85,B 0,C 180,E1 -15226.217,E2 -15226.217} C_VEL
LIN {X 0,Y 322.217,Z 576.612,A -85,B 0,C 180,E1 -15228.108,E2 -15228.108} C_VEL
LIN {X 0,Y 323.756,Z 565.338,A -85,B 0,C 180,E1 -15229.827,E2 -15229.827} C_VEL
LIN {X 0,Y 325.525,Z 552.922,A -85,B 0,C 180,E1 -15231.366,E2 -15231.366} C_VEL
LIN {X 0,Y 326.753,Z 541.019,A -85,B 0,C 180,E1 -15232.58,E2 -15232.58} C_VEL
LIN {X 0,Y 325.245,Z 527.838,A -85,B 0,C 180,E1 -15233.796,E2 -15233.796} C_VEL
LIN {X 0,Y 323.013,Z 512.839,A -85,B 0,C 180,E1 -15234.94,E2 -15234.94} C_VEL
LIN {X 0,Y 320.344,Z 497.55,A -85,B 0,C 180,E1 -15235.848,E2 -15235.848} C_VEL
LIN {X 0,Y 319.422,Z 492.273,A -85,B 0,C 180,E1 -15236.106,E2 -15236.106} C_VEL
LIN {X 0,Y 320.222,Z 485.137,A -85,B 0,C 180,E1 -15240.317,E2 -15240.317} C_VEL
LIN {X 0,Y 320.96,Z 479.551,A -85,B 0,C 180,E1 -15243.687,E2 -15243.687} C_VEL
LIN {X 0,Y 321.705,Z 474.328,A -85,B 0,C 180,E1 -15246.924,E2 -15246.924} C_VEL
LIN {X 0,Y 322.144,Z 470.663,A -85,B 0,C 180,E1 -15249.247,E2 -15249.247} C_VEL
LIN {X 0,Y 321.779,Z 466.515,A -85,B 0,C 180,E1 -15252.047,E2 -15252.047} C_VEL
LIN {X 0,Y 320.93,Z 461.646,A -85,B 0,C 180,E1 -15255.512,E2 -15255.512} C_VEL
LIN {X 0,Y 320.133,Z 457.267,A -85,B 0,C 180,E1 -15258.807,E2 -15258.807} C_VEL
LIN {X 0,Y 319.631,Z 454.298,A -85,B 0,C 180,E1 -15261.196,E2 -15261.196} C_VEL
LIN {X 0,Y 319.557,Z 454.307,A -85,B 0,C 180,E1 -15265.123,E2 -15265.123} C_VEL
LIN {X 0,Y 319.571,Z 454.305,A -85,B 0,C 180,E1 -15269.056,E2 -15269.056} C_VEL
LIN {X 0,Y 319.605,Z 454.297,A -85,B 0,C 180,E1 -15272.498,E2 -15272.498} C_VEL
LIN {X 0,Y 319.6,Z 454.298,A -85,B 0,C 180,E1 -15275.304,E2 -15275.304} C_VEL
LIN {X 0,Y 319.593,Z 454.297,A -85,B 0,C 180,E1 -15278.048,E2 -15278.048} C_VEL
LIN {X 0,Y 319.684,Z 454.29,A -85,B 0,C 180,E1 -15280.962,E2 -15280.962} C_VEL
LIN {X 0,Y 319.726,Z 454.282,A -85,B 0,C 180,E1 -15285.276,E2 -15285.276} C_VEL
LIN {X 0,Y 319.752,Z 454.277,A -85,B 0,C 180,E1 -15289.873,E2 -15289.873} C_VEL
LIN {X 0,Y 319.928,Z 454.258,A -85,B 0,C 180,E1 -15292.426,E2 -15292.426} C_VEL
LIN {X 0,Y 319.744,Z 454.281,A -85,B 0,C 180,E1 -15294.956,E2 -15294.956} C_VEL
LIN {X 0,Y 319.987,Z 454.248,A -85,B 0,C 180,E1 -15297.483,E2 -15297.483} C_VEL
LIN {X 0,Y 320.145,Z 454.229,A -85,B 0,C 180,E1 -15300,E2 -15300} C_VEL
LIN {X 0,Y 320.004,Z 454.251,A -85,B 0,C 180,E1 -15302.518,E2 -15302.518} C_VEL
LIN {X 0,Y 319.932,Z 454.256,A -85,B 0,C 180,E1 -15306.587,E2 -15306.587} C_VEL
LIN {X 0,Y 319.753,Z 454.28,A -85,B 0,C 180,E1 -15310.128,E2 -15310.128} C_VEL
LIN {X 0,Y 319.726,Z 454.283,A -85,B 0,C 180,E1 -15314.724,E2 -15314.724} C_VEL
LIN {X 0,Y 319.685,Z 454.286,A -85,B 0,C 180,E1 -15319.038,E2 -15319.038} C_VEL
LIN {X 0,Y 319.566,Z 454.3,A -85,B 0,C 180,E1 -15323.32,E2 -15323.32} C_VEL
LIN {X 0,Y 319.631,Z 454.296,A -85,B 0,C 180,E1 -15326.089,E2 -15326.089} C_VEL
LIN {X 0,Y 319.585,Z 454.298,A -85,B 0,C 180,E1 -15328.934,E2 -15328.934} C_VEL
LIN {X 0,Y 319.529,Z 454.308,A -85,B 0,C 180,E1 -15331.863,E2 -15331.863} C_VEL
LIN {X 0,Y 319.577,Z 454.3,A -85,B 0,C 180,E1 -15335.544,E2 -15335.544} C_VEL
LIN {X 0,Y 319.571,Z 454.305,A -85,B 0,C 180,E1 -15338.009,E2 -15338.009} C_VEL
LIN {X 0,Y 319.524,Z 454.307,A -85,B 0,C 180,E1 -15341.598,E2 -15341.598} C_VEL
LIN {X 0,Y 319.493,Z 454.31,A -85,B 0,C 180,E1 -15345.259,E2 -15345.259} C_VEL
LIN {X 0,Y 319.568,Z 454.302,A -85,B 0,C 180,E1 -15348.395,E2 -15348.395} C_VEL
LIN {X 0,Y 319.582,Z 454.3,A -85,B 0,C 180,E1 -15352.344,E2 -15352.344} C_VEL
LIN {X 0,Y 319.561,Z 454.301,A -85,B 0,C 180,E1 -15355.124,E2 -15355.124} C_VEL
LIN {X 0,Y 319.571,Z 454.3,A -85,B 0,C 180,E1 -15359.059,E2 -15359.059} C_VEL
LIN {X 0,Y 319.619,Z 454.294,A -85,B 0,C 180,E1 -15362.5,E2 -15362.5} C_VEL
LIN {X 0,Y 319.607,Z 454.297,A -85,B 0,C 180,E1 -15365.305,E2 -15365.305} C_VEL
LIN {X 0,Y 319.599,Z 454.299,A -85,B 0,C 180,E1 -15368.048,E2 -15368.048} C_VEL
LIN {X 0,Y 319.692,Z 454.285,A -85,B 0,C 180,E1 -15370.962,E2 -15370.962} C_VEL
LIN {X 0,Y 319.734,Z 454.282,A -85,B 0,C 180,E1 -15375.276,E2 -15375.276} C_VEL
LIN {X 0,Y 319.755,Z 454.279,A -85,B 0,C 180,E1 -15379.873,E2 -15379.873} C_VEL
LIN {X 0,Y 319.912,Z 454.261,A -85,B 0,C 180,E1 -15383.694,E2 -15383.694} C_VEL
LIN {X 0,Y 319.994,Z 454.252,A -85,B 0,C 180,E1 -15387.482,E2 -15387.482} C_VEL
LIN {X 0,Y 320.153,Z 454.228,A -85,B 0,C 180,E1 -15390,E2 -15390} C_VEL
LIN {X 0,Y 319.993,Z 454.247,A -85,B 0,C 180,E1 -15392.518,E2 -15392.518} C_VEL
LIN {X 0,Y 319.946,Z 454.253,A -85,B 0,C 180,E1 -15396.305,E2 -15396.305} C_VEL
LIN {X 0,Y 319.84,Z 454.268,A -85,B 0,C 180,E1 -15398.848,E2 -15398.848} C_VEL
LIN {X 0,Y 319.685,Z 454.287,A -85,B 0,C 180,E1 -15402.699,E2 -15402.699} C_VEL
LIN {X 0,Y 319.702,Z 454.288,A -85,B 0,C 180,E1 -15405.295,E2 -15405.295} C_VEL
LIN {X 0,Y 319.677,Z 454.291,A -85,B 0,C 180,E1 -15409.254,E2 -15409.254} C_VEL
LIN {X 0,Y 319.572,Z 454.303,A -85,B 0,C 180,E1 -15413.319,E2 -15413.319} C_VEL
LIN {X 0,Y 319.636,Z 454.292,A -85,B 0,C 180,E1 -15416.087,E2 -15416.087} C_VEL
LIN {X 0,Y 319.591,Z 454.302,A -85,B 0,C 180,E1 -15418.933,E2 -15418.933} C_VEL
LIN {X 0,Y 319.529,Z 454.305,A -85,B 0,C 180,E1 -15421.861,E2 -15421.861} C_VEL
LIN {X 0,Y 319.427,Z 454.323,A -85,B 0,C 180,E1 -15424.893,E2 -15424.893} C_VEL
LIN {X 0,Y 319.079,Z 454.361,A -85,B 0,C 180,E1 -15428.077,E2 -15428.077} C_VEL
LIN {X 0,Y 318.697,Z 454.414,A -85,B 0,C 180,E1 -15431.428,E2 -15431.428} C_VEL
LIN {X 0,Y 318.519,Z 454.993,A -85,B 0,C 180,E1 -15433.269,E2 -15433.269} C_VEL
LIN {X 0,Y 318.456,Z 457.2,A -85,B 0,C 180,E1 -15436.015,E2 -15436.015} C_VEL
LIN {X 0,Y 323.003,Z 473.126,A -85,B 0,C 180,E1 -15437.059,E2 -15437.059} C_VEL
LIN {X 0,Y 326.485,Z 486.552,A -85,B 0,C 180,E1 -15438.139,E2 -15438.139} C_VEL
LIN {X 0,Y 328.504,Z 495.338,A -85,B 0,C 180,E1 -15438.957,E2 -15438.957} C_VEL
LIN {X 0,Y 327.376,Z 507.631,A -85,B 0,C 180,E1 -15440.061,E2 -15440.061} C_VEL
LIN {X 0,Y 325.802,Z 520.461,A -85,B 0,C 180,E1 -15441.473,E2 -15441.473} C_VEL
LIN {X 0,Y 324.269,Z 532.603,A -85,B 0,C 180,E1 -15443.122,E2 -15443.122} C_VEL
LIN {X 0,Y 322.911,Z 542.652,A -85,B 0,C 180,E1 -15444.777,E2 -15444.777} C_VEL
LIN {X 0,Y 321.787,Z 551.153,A -85,B 0,C 180,E1 -15446.448,E2 -15446.448} C_VEL
LIN {X 0,Y 320.627,Z 558.945,A -85,B 0,C 180,E1 -15448.259,E2 -15448.259} C_VEL
LIN {X 0,Y 319.718,Z 566.404,A -85,B 0,C 180,E1 -15450.357,E2 -15450.357} C_VEL
LIN {X 0,Y 319.041,Z 572.431,A -85,B 0,C 180,E1 -15452.445,E2 -15452.445} C_VEL
LIN {X 0,Y 318.48,Z 577.779,A -85,B 0,C 180,E1 -15454.789,E2 -15454.789} C_VEL
LIN {X 0,Y 318.231,Z 580.077,A -85,B 0,C 180,E1 -15456.057,E2 -15456.057} C_VEL
LIN {X 0,Y 317.394,Z 581.708,A -85,B 0,C 180,E1 -15457.071,E2 -15457.071} C_VEL
LIN {X 0,Y 314.313,Z 583.923,A -85,B 0,C 180,E1 -15458.734,E2 -15458.734} C_VEL
LIN {X 0,Y 311.81,Z 585.282,A -85,B 0,C 180,E1 -15460.097,E2 -15460.097} C_VEL
LIN {X 0,Y 310.783,Z 586.059,A -85,B 0,C 180,E1 -15461.162,E2 -15461.162} C_VEL
LIN {X 0,Y 310.72,Z 586.225,A -85,B 0,C 180,E1 -15461.524,E2 -15461.524} C_VEL
LIN {X 0,Y 310.785,Z 586.707,A -85,B 0,C 180,E1 -15462.903,E2 -15462.903} C_VEL
LIN {X 0,Y 311.024,Z 586.55,A -85,B 0,C 180,E1 -15465.607,E2 -15465.607} C_VEL
LIN {X 0,Y 311.522,Z 584.965,A -85,B 0,C 180,E1 -15468.285,E2 -15468.285} C_VEL
LIN {X 0,Y 312.352,Z 581.951,A -85,B 0,C 180,E1 -15470.938,E2 -15470.938} C_VEL
LIN {X 0,Y 313.477,Z 577.444,A -85,B 0,C 180,E1 -15473.563,E2 -15473.563} C_VEL
LIN {X 0,Y 315.135,Z 571.315,A -85,B 0,C 180,E1 -15476.164,E2 -15476.164} C_VEL
LIN {X 0,Y 316.79,Z 565.132,A -85,B 0,C 180,E1 -15478.234,E2 -15478.234} C_VEL
LIN {X 0,Y 318.699,Z 557.539,A -85,B 0,C 180,E1 -15480.316,E2 -15480.316} C_VEL
LIN {X 0,Y 320.896,Z 549.114,A -85,B 0,C 180,E1 -15482.196,E2 -15482.196} C_VEL
LIN {X 0,Y 323.645,Z 537.929,A -85,B 0,C 180,E1 -15484.249,E2 -15484.249} C_VEL
LIN {X 0,Y 325.991,Z 527.553,A -85,B 0,C 180,E1 -15485.807,E2 -15485.807} C_VEL
LIN {X 0,Y 328.569,Z 514.743,A -85,B 0,C 180,E1 -15487.373,E2 -15487.373} C_VEL
LIN {X 0,Y 330.006,Z 506.645,A -85,B 0,C 180,E1 -15488.207,E2 -15488.207} C_VEL
LIN {X 0,Y 328.317,Z 498.231,A -85,B 0,C 180,E1 -15489.415,E2 -15489.415} C_VEL
LIN {X 0,Y 324.875,Z 488.194,A -85,B 0,C 180,E1 -15490.956,E2 -15490.956} C_VEL
LIN {X 0,Y 320.104,Z 477.801,A -85,B 0,C 180,E1 -15492.683,E2 -15492.683} C_VEL
LIN {X 0,Y 317.661,Z 473.446,A -85,B 0,C 180,E1 -15493.49,E2 -15493.49} C_VEL
LIN {X 0,Y 315.603,Z 469.723,A -85,B 0,C 180,E1 -15494.179,E2 -15494.179} C_VEL
LIN {X 0,Y 313.871,Z 467.161,A -85,B 0,C 180,E1 -15494.703,E2 -15494.703} C_VEL
LIN {X 0,Y 313.343,Z 465.347,A -85,B 0,C 180,E1 -15494.976,E2 -15494.976} C_VEL
LIN {X 0,Y 313.626,Z 464.396,A -85,B 0,C 180,E1 -15498.284,E2 -15498.284} C_VEL
LIN {X 0,Y 313.777,Z 463.836,A -85,B 0,C 180,E1 -15501,E2 -15501} C_VEL
LIN {X 0,Y 313.839,Z 463.522,A -85,B 0,C 180,E1 -15503.771,E2 -15503.771} C_VEL
LIN {X 0,Y 313.938,Z 463.456,A -85,B 0,C 180,E1 -15506.598,E2 -15506.598} C_VEL
LIN {X 0,Y 313.983,Z 463.688,A -85,B 0,C 180,E1 -15509.501,E2 -15509.501} C_VEL
LIN {X 0,Y 314.086,Z 464.288,A -85,B 0,C 180,E1 -15512.481,E2 -15512.481} C_VEL
LIN {X 0,Y 314.336,Z 465.626,A -85,B 0,C 180,E1 -15516.401,E2 -15516.401} C_VEL
LIN {X 0,Y 314.751,Z 467.657,A -85,B 0,C 180,E1 -15520.356,E2 -15520.356} C_VEL
LIN {X 0,Y 315.133,Z 469.976,A -85,B 0,C 180,E1 -15523.737,E2 -15523.737} C_VEL
LIN {X 0,Y 315.588,Z 473.009,A -85,B 0,C 180,E1 -15527.298,E2 -15527.298} C_VEL
LIN {X 0,Y 315.686,Z 475.536,A -85,B 0,C 180,E1 -15529.789,E2 -15529.789} C_VEL
LIN {X 0,Y 315.516,Z 477.368,A -85,B 0,C 180,E1 -15531.415,E2 -15531.415} C_VEL
LIN {X 0,Y 314.767,Z 481.267,A -85,B 0,C 180,E1 -15534.514,E2 -15534.514} C_VEL
LIN {X 0,Y 314.085,Z 484.959,A -85,B 0,C 180,E1 -15537.138,E2 -15537.138} C_VEL
LIN {X 0,Y 315.138,Z 488.568,A -85,B 0,C 180,E1 -15537.568,E2 -15537.568} C_VEL
LIN {X 0,Y 316.114,Z 490.639,A -85,B 0,C 180,E1 -15537.885,E2 -15537.885} C_VEL
LIN {X 0,Y 320.639,Z 504.348,A -85,B 0,C 180,E1 -15539.65,E2 -15539.65} C_VEL
LIN {X 0,Y 323.867,Z 518.543,A -85,B 0,C 180,E1 -15541.361,E2 -15541.361} C_VEL
LIN {X 0,Y 325.338,Z 530.123,A -85,B 0,C 180,E1 -15542.738,E2 -15542.738} C_VEL
LIN {X 0,Y 325.609,Z 541.729,A -85,B 0,C 180,E1 -15544.116,E2 -15544.116} C_VEL
LIN {X 0,Y 325.024,Z 549.466,A -85,B 0,C 180,E1 -15545.062,E2 -15545.062} C_VEL
LIN {X 0,Y 322.663,Z 559.82,A -85,B 0,C 180,E1 -15546.348,E2 -15546.348} C_VEL
LIN {X 0,Y 320.075,Z 571.385,A -85,B 0,C 180,E1 -15548.083,E2 -15548.083} C_VEL
LIN {X 0,Y 317.72,Z 581.674,A -85,B 0,C 180,E1 -15549.949,E2 -15549.949} C_VEL
LIN {X 0,Y 315.46,Z 591.647,A -85,B 0,C 180,E1 -15552.162,E2 -15552.162} C_VEL
LIN {X 0,Y 313.633,Z 600.145,A -85,B 0,C 180,E1 -15554.485,E2 -15554.485} C_VEL
LIN {X 0,Y 312.315,Z 607.508,A -85,B 0,C 180,E1 -15556.996,E2 -15556.996} C_VEL
LIN {X 0,Y 311.357,Z 613.444,A -85,B 0,C 180,E1 -15559.597,E2 -15559.597} C_VEL
LIN {X 0,Y 310.92,Z 617.852,A -85,B 0,C 180,E1 -15562.205,E2 -15562.205} C_VEL
LIN {X 0,Y 310.78,Z 620.807,A -85,B 0,C 180,E1 -15564.81,E2 -15564.81} C_VEL
LIN {X 0,Y 310.836,Z 621.754,A -85,B 0,C 180,E1 -15566.111,E2 -15566.111} C_VEL
LIN {X 0,Y 310.952,Z 622.593,A -85,B 0,C 180,E1 -15568.705,E2 -15568.705} C_VEL
LIN {X 0,Y 311.095,Z 622.49,A -85,B 0,C 180,E1 -15570,E2 -15570} C_VEL
LIN {X 0,Y 311.017,Z 622.016,A -85,B 0,C 180,E1 -15571.295,E2 -15571.295} C_VEL
LIN {X 0,Y 310.867,Z 619.984,A -85,B 0,C 180,E1 -15573.889,E2 -15573.889} C_VEL
LIN {X 0,Y 310.929,Z 617.278,A -85,B 0,C 180,E1 -15575.99,E2 -15575.99} C_VEL
LIN {X 0,Y 311.064,Z 612.771,A -85,B 0,C 180,E1 -15578.445,E2 -15578.445} C_VEL
LIN {X 0,Y 311.348,Z 608.123,A -85,B 0,C 180,E1 -15580.404,E2 -15580.404} C_VEL
LIN {X 0,Y 312.049,Z 601.339,A -85,B 0,C 180,E1 -15582.685,E2 -15582.685} C_VEL
LIN {X 0,Y 312.805,Z 593.572,A -85,B 0,C 180,E1 -15584.794,E2 -15584.794} C_VEL
LIN {X 0,Y 314.164,Z 584.024,A -85,B 0,C 180,E1 -15586.906,E2 -15586.906} C_VEL
LIN {X 0,Y 315.617,Z 573.376,A -85,B 0,C 180,E1 -15588.837,E2 -15588.837} C_VEL
LIN {X 0,Y 317.428,Z 561.597,A -85,B 0,C 180,E1 -15590.577,E2 -15590.577} C_VEL
LIN {X 0,Y 318.978,Z 549.878,A -85,B 0,C 180,E1 -15591.997,E2 -15591.997} C_VEL
LIN {X 0,Y 319.856,Z 542.05,A -85,B 0,C 180,E1 -15592.797,E2 -15592.797} C_VEL
LIN {X 0,Y 318.379,Z 528.866,A -85,B 0,C 180,E1 -15594.071,E2 -15594.071} C_VEL
LIN {X 0,Y 316.339,Z 514.705,A -85,B 0,C 180,E1 -15595.207,E2 -15595.207} C_VEL
LIN {X 0,Y 313.802,Z 499.553,A -85,B 0,C 180,E1 -15596.178,E2 -15596.178} C_VEL
LIN {X 0,Y 312.43,Z 491.846,A -85,B 0,C 180,E1 -15596.605,E2 -15596.605} C_VEL
LIN {X 0,Y 313.312,Z 484.517,A -85,B 0,C 180,E1 -15601.058,E2 -15601.058} C_VEL
LIN {X 0,Y 314.135,Z 478.54,A -85,B 0,C 180,E1 -15604.784,E2 -15604.784} C_VEL
LIN {X 0,Y 314.839,Z 473.709,A -85,B 0,C 180,E1 -15607.869,E2 -15607.869} C_VEL
LIN {X 0,Y 315.063,Z 470.038,A -85,B 0,C 180,E1 -15610.307,E2 -15610.307} C_VEL
LIN {X 0,Y 314.651,Z 466.872,A -85,B 0,C 180,E1 -15612.517,E2 -15612.517} C_VEL
LIN {X 0,Y 313.761,Z 462.102,A -85,B 0,C 180,E1 -15616.023,E2 -15616.023} C_VEL
LIN {X 0,Y 312.925,Z 457.242,A -85,B 0,C 180,E1 -15619.782,E2 -15619.782} C_VEL
LIN {X 0,Y 312.584,Z 455.175,A -85,B 0,C 180,E1 -15621.502,E2 -15621.502} C_VEL
LIN {X 0,Y 312.528,Z 455.178,A -85,B 0,C 180,E1 -15624.22,E2 -15624.22} C_VEL
LIN {X 0,Y 312.503,Z 455.183,A -85,B 0,C 180,E1 -15627.334,E2 -15627.334} C_VEL
LIN {X 0,Y 312.549,Z 455.177,A -85,B 0,C 180,E1 -15631.276,E2 -15631.276} C_VEL
LIN {X 0,Y 312.581,Z 455.173,A -85,B 0,C 180,E1 -15634.711,E2 -15634.711} C_VEL
LIN {X 0,Y 312.583,Z 455.171,A -85,B 0,C 180,E1 -15637.529,E2 -15637.529} C_VEL
LIN {X 0,Y 312.633,Z 455.164,A -85,B 0,C 180,E1 -15641.656,E2 -15641.656} C_VEL
LIN {X 0,Y 312.689,Z 455.157,A -85,B 0,C 180,E1 -15645.686,E2 -15645.686} C_VEL
LIN {X 0,Y 312.697,Z 455.156,A -85,B 0,C 180,E1 -15649.642,E2 -15649.642} C_VEL
LIN {X 0,Y 312.866,Z 455.136,A -85,B 0,C 180,E1 -15652.254,E2 -15652.254} C_VEL
LIN {X 0,Y 312.714,Z 455.158,A -85,B 0,C 180,E1 -15654.843,E2 -15654.843} C_VEL
LIN {X 0,Y 312.988,Z 455.124,A -85,B 0,C 180,E1 -15658.714,E2 -15658.714} C_VEL
LIN {X 0,Y 312.987,Z 455.12,A -85,B 0,C 180,E1 -15661.287,E2 -15661.287} C_VEL
LIN {X 0,Y 312.694,Z 455.157,A -85,B 0,C 180,E1 -15663.866,E2 -15663.866} C_VEL
LIN {X 0,Y 312.898,Z 455.135,A -85,B 0,C 180,E1 -15666.569,E2 -15666.569} C_VEL
LIN {X 0,Y 312.783,Z 455.146,A -85,B 0,C 180,E1 -15669.05,E2 -15669.05} C_VEL
LIN {X 0,Y 312.63,Z 455.165,A -85,B 0,C 180,E1 -15672.992,E2 -15672.992} C_VEL
LIN {X 0,Y 312.634,Z 455.164,A -85,B 0,C 180,E1 -15675.65,E2 -15675.65} C_VEL
LIN {X 0,Y 312.627,Z 455.164,A -85,B 0,C 180,E1 -15679.237,E2 -15679.237} C_VEL
LIN {X 0,Y 312.542,Z 455.177,A -85,B 0,C 180,E1 -15682.79,E2 -15682.79} C_VEL
LIN {X 0,Y 312.599,Z 455.171,A -85,B 0,C 180,E1 -15685.936,E2 -15685.936} C_VEL
LIN {X 0,Y 312.542,Z 455.176,A -85,B 0,C 180,E1 -15689.651,E2 -15689.651} C_VEL
LIN {X 0,Y 312.517,Z 455.18,A -85,B 0,C 180,E1 -15693.69,E2 -15693.69} C_VEL
LIN {X 0,Y 312.523,Z 455.178,A -85,B 0,C 180,E1 -15697.386,E2 -15697.386} C_VEL
LIN {X 0,Y 312.488,Z 455.183,A -85,B 0,C 180,E1 -15700.71,E2 -15700.71} C_VEL
LIN {X 0,Y 312.452,Z 455.19,A -85,B 0,C 180,E1 -15704.21,E2 -15704.21} C_VEL
LIN {X 0,Y 312.527,Z 455.182,A -85,B 0,C 180,E1 -15707.911,E2 -15707.911} C_VEL
LIN {X 0,Y 312.556,Z 455.179,A -85,B 0,C 180,E1 -15711.906,E2 -15711.906} C_VEL
LIN {X 0,Y 312.507,Z 455.184,A -85,B 0,C 180,E1 -15715.791,E2 -15715.791} C_VEL
LIN {X 0,Y 312.525,Z 455.177,A -85,B 0,C 180,E1 -15718.855,E2 -15718.855} C_VEL
LIN {X 0,Y 312.586,Z 455.175,A -85,B 0,C 180,E1 -15721.827,E2 -15721.827} C_VEL
LIN {X 0,Y 312.587,Z 455.169,A -85,B 0,C 180,E1 -15724.712,E2 -15724.712} C_VEL
LIN {X 0,Y 312.589,Z 455.173,A -85,B 0,C 180,E1 -15727.53,E2 -15727.53} C_VEL
LIN {X 0,Y 312.641,Z 455.168,A -85,B 0,C 180,E1 -15731.657,E2 -15731.657} C_VEL
LIN {X 0,Y 312.697,Z 455.161,A -85,B 0,C 180,E1 -15735.687,E2 -15735.687} C_VEL
LIN {X 0,Y 312.701,Z 455.16,A -85,B 0,C 180,E1 -15739.642,E2 -15739.642} C_VEL
LIN {X 0,Y 312.806,Z 455.143,A -85,B 0,C 180,E1 -15742.253,E2 -15742.253} C_VEL
LIN {X 0,Y 312.71,Z 455.155,A -85,B 0,C 180,E1 -15744.842,E2 -15744.842} C_VEL
LIN {X 0,Y 312.94,Z 455.131,A -85,B 0,C 180,E1 -15747.426,E2 -15747.426} C_VEL
LIN {X 0,Y 313.105,Z 455.106,A -85,B 0,C 180,E1 -15750,E2 -15750} C_VEL
LIN {X 0,Y 312.94,Z 455.126,A -85,B 0,C 180,E1 -15752.574,E2 -15752.574} C_VEL
LIN {X 0,Y 312.903,Z 455.13,A -85,B 0,C 180,E1 -15756.448,E2 -15756.448} C_VEL
LIN {X 0,Y 312.77,Z 455.15,A -85,B 0,C 180,E1 -15759.05,E2 -15759.05} C_VEL
LIN {X 0,Y 312.638,Z 455.167,A -85,B 0,C 180,E1 -15762.991,E2 -15762.991} C_VEL
LIN {X 0,Y 312.641,Z 455.165,A -85,B 0,C 180,E1 -15765.649,E2 -15765.649} C_VEL
LIN {X 0,Y 312.633,Z 455.169,A -85,B 0,C 180,E1 -15769.236,E2 -15769.236} C_VEL
LIN {X 0,Y 312.548,Z 455.177,A -85,B 0,C 180,E1 -15772.789,E2 -15772.789} C_VEL
LIN {X 0,Y 312.604,Z 455.168,A -85,B 0,C 180,E1 -15775.935,E2 -15775.935} C_VEL
LIN {X 0,Y 312.546,Z 455.176,A -85,B 0,C 180,E1 -15779.649,E2 -15779.649} C_VEL
LIN {X 0,Y 312.471,Z 455.187,A -85,B 0,C 180,E1 -15782.669,E2 -15782.669} C_VEL
LIN {X 0,Y 312.273,Z 455.209,A -85,B 0,C 180,E1 -15785.882,E2 -15785.882} C_VEL
LIN {X 0,Y 311.909,Z 455.259,A -85,B 0,C 180,E1 -15789.116,E2 -15789.116} C_VEL
LIN {X 0,Y 311.48,Z 455.313,A -85,B 0,C 180,E1 -15792.601,E2 -15792.601} C_VEL
LIN {X 0,Y 311.405,Z 457.688,A -85,B 0,C 180,E1 -15795.577,E2 -15795.577} C_VEL
LIN {X 0,Y 315.841,Z 473.224,A -85,B 0,C 180,E1 -15796.606,E2 -15796.606} C_VEL
LIN {X 0,Y 319.359,Z 486.613,A -85,B 0,C 180,E1 -15797.706,E2 -15797.706} C_VEL
LIN {X 0,Y 321.68,Z 496.702,A -85,B 0,C 180,E1 -15798.676,E2 -15798.676} C_VEL
LIN {X 0,Y 320.45,Z 509.277,A -85,B 0,C 180,E1 -15799.849,E2 -15799.849} C_VEL
LIN {X 0,Y 318.831,Z 521.826,A -85,B 0,C 180,E1 -15801.283,E2 -15801.283} C_VEL
LIN {X 0,Y 317.235,Z 533.895,A -85,B 0,C 180,E1 -15802.981,E2 -15802.981} C_VEL
LIN {X 0,Y 315.695,Z 545.043,A -85,B 0,C 180,E1 -15804.914,E2 -15804.914} C_VEL
LIN {X 0,Y 314.4,Z 554.019,A -85,B 0,C 180,E1 -15806.793,E2 -15806.793} C_VEL
LIN {X 0,Y 313.229,Z 562.441,A -85,B 0,C 180,E1 -15808.931,E2 -15808.931} C_VEL
LIN {X 0,Y 312.324,Z 570.112,A -85,B 0,C 180,E1 -15811.351,E2 -15811.351} C_VEL
LIN {X 0,Y 311.568,Z 576.447,A -85,B 0,C 180,E1 -15813.905,E2 -15813.905} C_VEL
LIN {X 0,Y 311.144,Z 580.416,A -85,B 0,C 180,E1 -15816.01,E2 -15816.01} C_VEL
LIN {X 0,Y 310.891,Z 583.174,A -85,B 0,C 180,E1 -15817.946,E2 -15817.946} C_VEL
LIN {X 0,Y 310.718,Z 585.386,A -85,B 0,C 180,E1 -15820.167,E2 -15820.167} C_VEL
LIN {X 0,Y 310.72,Z 586.225,A -85,B 0,C 180,E1 -15821.524,E2 -15821.524} C_VEL
LIN {X 0,Y 310.125,Z 586.777,A -85,B 0,C 180,E1 -15822.603,E2 -15822.603} C_VEL
LIN {X 0,Y 307.393,Z 587.16,A -85,B 0,C 180,E1 -15824.371,E2 -15824.371} C_VEL
LIN {X 0,Y 305.121,Z 586.97,A -85,B 0,C 180,E1 -15825.805,E2 -15825.805} C_VEL
LIN {X 0,Y 304.243,Z 586.561,A -85,B 0,C 180,E1 -15826.91,E2 -15826.91} C_VEL
LIN {X 0,Y 304.224,Z 586.322,A -85,B 0,C 180,E1 -15827.282,E2 -15827.282} C_VEL
LIN {X 0,Y 304.751,Z 584.719,A -85,B 0,C 180,E1 -15829.368,E2 -15829.368} C_VEL
LIN {X 0,Y 305.77,Z 581.304,A -85,B 0,C 180,E1 -15832.073,E2 -15832.073} C_VEL
LIN {X 0,Y 307.136,Z 576.429,A -85,B 0,C 180,E1 -15834.748,E2 -15834.748} C_VEL
LIN {X 0,Y 308.525,Z 571.664,A -85,B 0,C 180,E1 -15836.735,E2 -15836.735} C_VEL
LIN {X 0,Y 310.416,Z 564.885,A -85,B 0,C 180,E1 -15839.027,E2 -15839.027} C_VEL
LIN {X 0,Y 312.738,Z 556.546,A -85,B 0,C 180,E1 -15841.287,E2 -15841.287} C_VEL
LIN {X 0,Y 315.134,Z 547.912,A -85,B 0,C 180,E1 -15843.196,E2 -15843.196} C_VEL
LIN {X 0,Y 317.785,Z 537.576,A -85,B 0,C 180,E1 -15845.075,E2 -15845.075} C_VEL
LIN {X 0,Y 320.508,Z 526.118,A -85,B 0,C 180,E1 -15846.768,E2 -15846.768} C_VEL
LIN {X 0,Y 323.042,Z 514.213,A -85,B 0,C 180,E1 -15848.227,E2 -15848.227} C_VEL
LIN {X 0,Y 324.031,Z 509.385,A -85,B 0,C 180,E1 -15848.732,E2 -15848.732} C_VEL
LIN {X 0,Y 322.891,Z 502.395,A -85,B 0,C 180,E1 -15849.77,E2 -15849.77} C_VEL
LIN {X 0,Y 320.075,Z 493.181,A -85,B 0,C 180,E1 -15851.267,E2 -15851.267} C_VEL
LIN {X 0,Y 315.811,Z 483.138,A -85,B 0,C 180,E1 -15853.038,E2 -15853.038} C_VEL
LIN {X 0,Y 311.229,Z 474.723,A -85,B 0,C 180,E1 -15854.698,E2 -15854.698} C_VEL
LIN {X 0,Y 309.575,Z 471.661,A -85,B 0,C 180,E1 -15855.33,E2 -15855.33} C_VEL
LIN {X 0,Y 308.649,Z 470.416,A -85,B 0,C 180,E1 -15855.637,E2 -15855.637} C_VEL
LIN {X 0,Y 306.934,Z 467.851,A -85,B 0,C 180,E1 -15856.229,E2 -15856.229} C_VEL
LIN {X 0,Y 306.46,Z 466.253,A -85,B 0,C 180,E1 -15856.478,E2 -15856.478} C_VEL
LIN {X 0,Y 306.821,Z 465.414,A -85,B 0,C 180,E1 -15860.095,E2 -15860.095} C_VEL
LIN {X 0,Y 306.904,Z 464.998,A -85,B 0,C 180,E1 -15863.656,E2 -15863.656} C_VEL
LIN {X 0,Y 306.993,Z 464.988,A -85,B 0,C 180,E1 -15867.249,E2 -15867.249} C_VEL
LIN {X 0,Y 307.062,Z 465.357,A -85,B 0,C 180,E1 -15870.234,E2 -15870.234} C_VEL
LIN {X 0,Y 307.183,Z 466.062,A -85,B 0,C 180,E1 -15873.305,E2 -15873.305} C_VEL
LIN {X 0,Y 307.461,Z 467.377,A -85,B 0,C 180,E1 -15876.868,E2 -15876.868} C_VEL
LIN {X 0,Y 307.73,Z 468.845,A -85,B 0,C 180,E1 -15879.752,E2 -15879.752} C_VEL
LIN {X 0,Y 308.134,Z 471.056,A -85,B 0,C 180,E1 -15883.176,E2 -15883.176} C_VEL
LIN {X 0,Y 308.586,Z 474.099,A -85,B 0,C 180,E1 -15886.903,E2 -15886.903} C_VEL
LIN {X 0,Y 308.702,Z 475.802,A -85,B 0,C 180,E1 -15888.702,E2 -15888.702} C_VEL
LIN {X 0,Y 308.596,Z 477.964,A -85,B 0,C 180,E1 -15890.743,E2 -15890.743} C_VEL
LIN {X 0,Y 307.993,Z 481.368,A -85,B 0,C 180,E1 -15893.61,E2 -15893.61} C_VEL
LIN {X 0,Y 307.415,Z 484.011,A -85,B 0,C 180,E1 -15895.661,E2 -15895.661} C_VEL
LIN {X 0,Y 308.396,Z 487.611,A -85,B 0,C 180,E1 -15896.14,E2 -15896.14} C_VEL
LIN {X 0,Y 309.66,Z 490.246,A -85,B 0,C 180,E1 -15896.599,E2 -15896.599} C_VEL
LIN {X 0,Y 313.135,Z 500.042,A -85,B 0,C 180,E1 -15898.012,E2 -15898.012} C_VEL
LIN {X 0,Y 316.145,Z 510.926,A -85,B 0,C 180,E1 -15899.477,E2 -15899.477} C_VEL
LIN {X 0,Y 318.413,Z 523.395,A -85,B 0,C 180,E1 -15901.071,E2 -15901.071} C_VEL
LIN {X 0,Y 319.412,Z 534.683,A -85,B 0,C 180,E1 -15902.48,E2 -15902.48} C_VEL
LIN {X 0,Y 319.273,Z 545.634,A -85,B 0,C 180,E1 -15903.881,E2 -15903.881} C_VEL
LIN {X 0,Y 318.698,Z 550.762,A -85,B 0,C 180,E1 -15904.532,E2 -15904.532} C_VEL
LIN {X 0,Y 315.841,Z 562.636,A -85,B 0,C 180,E1 -15906.097,E2 -15906.097} C_VEL
LIN {X 0,Y 313.104,Z 573.862,A -85,B 0,C 180,E1 -15907.916,E2 -15907.916} C_VEL
LIN {X 0,Y 310.336,Z 585.096,A -85,B 0,C 180,E1 -15910.142,E2 -15910.142} C_VEL
LIN {X 0,Y 308.105,Z 594.413,A -85,B 0,C 180,E1 -15912.408,E2 -15912.408} C_VEL
LIN {X 0,Y 306.301,Z 602.801,A -85,B 0,C 180,E1 -15914.969,E2 -15914.969} C_VEL
LIN {X 0,Y 305.059,Z 609.08,A -85,B 0,C 180,E1 -15917.358,E2 -15917.358} C_VEL
LIN {X 0,Y 304.162,Z 614.5,A -85,B 0,C 180,E1 -15920.021,E2 -15920.021} C_VEL
LIN {X 0,Y 303.843,Z 617.611,A -85,B 0,C 180,E1 -15922.023,E2 -15922.023} C_VEL
LIN {X 0,Y 303.685,Z 620.459,A -85,B 0,C 180,E1 -15924.689,E2 -15924.689} C_VEL
LIN {X 0,Y 303.74,Z 621.368,A -85,B 0,C 180,E1 -15926.02,E2 -15926.02} C_VEL
LIN {X 0,Y 303.859,Z 622.134,A -85,B 0,C 180,E1 -15928.675,E2 -15928.675} C_VEL
LIN {X 0,Y 304.02,Z 621.994,A -85,B 0,C 180,E1 -15930,E2 -15930} C_VEL
LIN {X 0,Y 303.926,Z 621.481,A -85,B 0,C 180,E1 -15931.325,E2 -15931.325} C_VEL
LIN {X 0,Y 303.8,Z 619.371,A -85,B 0,C 180,E1 -15933.98,E2 -15933.98} C_VEL
LIN {X 0,Y 303.855,Z 616.831,A -85,B 0,C 180,E1 -15935.976,E2 -15935.976} C_VEL
LIN {X 0,Y 303.952,Z 613.372,A -85,B 0,C 180,E1 -15937.974,E2 -15937.974} C_VEL
LIN {X 0,Y 304.188,Z 608.947,A -85,B 0,C 180,E1 -15939.978,E2 -15939.978} C_VEL
LIN {X 0,Y 304.849,Z 602.506,A -85,B 0,C 180,E1 -15942.313,E2 -15942.313} C_VEL
LIN {X 0,Y 305.633,Z 594.439,A -85,B 0,C 180,E1 -15944.652,E2 -15944.652} C_VEL
LIN {X 0,Y 306.849,Z 586.042,A -85,B 0,C 180,E1 -15946.636,E2 -15946.636} C_VEL
LIN {X 0,Y 308.295,Z 575.949,A -85,B 0,C 180,E1 -15948.611,E2 -15948.611} C_VEL
LIN {X 0,Y 309.94,Z 564.73,A -85,B 0,C 180,E1 -15950.403,E2 -15950.403} C_VEL
LIN {X 0,Y 311.79,Z 552.371,A -85,B 0,C 180,E1 -15952.008,E2 -15952.008} C_VEL
LIN {X 0,Y 312.912,Z 542.664,A -85,B 0,C 180,E1 -15953.068,E2 -15953.068} C_VEL
LIN {X 0,Y 311.51,Z 529.667,A -85,B 0,C 180,E1 -15954.372,E2 -15954.372} C_VEL
LIN {X 0,Y 309.484,Z 515.329,A -85,B 0,C 180,E1 -15955.56,E2 -15955.56} C_VEL
LIN {X 0,Y 306.895,Z 499.774,A -85,B 0,C 180,E1 -15956.59,E2 -15956.59} C_VEL
LIN {X 0,Y 305.415,Z 491.564,A -85,B 0,C 180,E1 -15957.042,E2 -15957.042} C_VEL
LIN {X 0,Y 306.231,Z 485.074,A -85,B 0,C 180,E1 -15961.089,E2 -15961.089} C_VEL
LIN {X 0,Y 307.095,Z 479.107,A -85,B 0,C 180,E1 -15964.899,E2 -15964.899} C_VEL
LIN {X 0,Y 307.831,Z 474.294,A -85,B 0,C 180,E1 -15968.055,E2 -15968.055} C_VEL
LIN {X 0,Y 308.016,Z 470.832,A -85,B 0,C 180,E1 -15970.401,E2 -15970.401} C_VEL
LIN {X 0,Y 307.416,Z 466.824,A -85,B 0,C 180,E1 -15973.301,E2 -15973.301} C_VEL
LIN {X 0,Y 306.473,Z 461.683,A -85,B 0,C 180,E1 -15977.206,E2 -15977.206} C_VEL
LIN {X 0,Y 305.886,Z 458.235,A -85,B 0,C 180,E1 -15979.96,E2 -15979.96} C_VEL
LIN {X 0,Y 305.553,Z 456.052,A -85,B 0,C 180,E1 -15981.819,E2 -15981.819} C_VEL
LIN {X 0,Y 305.461,Z 456.057,A -85,B 0,C 180,E1 -15985.921,E2 -15985.921} C_VEL
LIN {X 0,Y 305.462,Z 456.059,A -85,B 0,C 180,E1 -15989.591,E2 -15989.591} C_VEL
LIN {X 0,Y 305.517,Z 456.053,A -85,B 0,C 180,E1 -15992.608,E2 -15992.608} C_VEL
LIN {X 0,Y 305.503,Z 456.053,A -85,B 0,C 180,E1 -15995.539,E2 -15995.539} C_VEL
LIN {X 0,Y 305.515,Z 456.051,A -85,B 0,C 180,E1 -15999.815,E2 -15999.815} C_VEL
LIN {X 0,Y 305.569,Z 456.047,A -85,B 0,C 180,E1 -16002.603,E2 -16002.603} C_VEL
LIN {X 0,Y 305.644,Z 456.036,A -85,B 0,C 180,E1 -16005.349,E2 -16005.349} C_VEL
LIN {X 0,Y 305.633,Z 456.037,A -85,B 0,C 180,E1 -16009.4,E2 -16009.4} C_VEL
LIN {X 0,Y 305.807,Z 456.015,A -85,B 0,C 180,E1 -16012.074,E2 -16012.074} C_VEL
LIN {X 0,Y 305.685,Z 456.035,A -85,B 0,C 180,E1 -16014.724,E2 -16014.724} C_VEL
LIN {X 0,Y 305.954,Z 456.001,A -85,B 0,C 180,E1 -16018.684,E2 -16018.684} C_VEL
LIN {X 0,Y 305.954,Z 455.996,A -85,B 0,C 180,E1 -16021.317,E2 -16021.317} C_VEL
LIN {X 0,Y 305.689,Z 456.029,A -85,B 0,C 180,E1 -16025.277,E2 -16025.277} C_VEL
LIN {X 0,Y 305.809,Z 456.015,A -85,B 0,C 180,E1 -16027.926,E2 -16027.926} C_VEL
LIN {X 0,Y 305.599,Z 456.041,A -85,B 0,C 180,E1 -16031.946,E2 -16031.946} C_VEL
LIN {X 0,Y 305.633,Z 456.037,A -85,B 0,C 180,E1 -16035.035,E2 -16035.035} C_VEL
LIN {X 0,Y 305.573,Z 456.043,A -85,B 0,C 180,E1 -16039.446,E2 -16039.446} C_VEL
LIN {X 0,Y 305.487,Z 456.055,A -85,B 0,C 180,E1 -16043.042,E2 -16043.042} C_VEL
LIN {X 0,Y 305.544,Z 456.052,A -85,B 0,C 180,E1 -16046.228,E2 -16046.228} C_VEL
LIN {X 0,Y 305.492,Z 456.053,A -85,B 0,C 180,E1 -16049.05,E2 -16049.05} C_VEL
LIN {X 0,Y 305.441,Z 456.063,A -85,B 0,C 180,E1 -16051.953,E2 -16051.953} C_VEL
LIN {X 0,Y 305.46,Z 456.057,A -85,B 0,C 180,E1 -16055.114,E2 -16055.114} C_VEL
LIN {X 0,Y 305.465,Z 456.059,A -85,B 0,C 180,E1 -16058.534,E2 -16058.534} C_VEL
LIN {X 0,Y 305.454,Z 456.059,A -85,B 0,C 180,E1 -16062.587,E2 -16062.587} C_VEL
LIN {X 0,Y 305.486,Z 456.055,A -85,B 0,C 180,E1 -16067.409,E2 -16067.409} C_VEL
LIN {X 0,Y 305.518,Z 456.053,A -85,B 0,C 180,E1 -16071.605,E2 -16071.605} C_VEL
LIN {X 0,Y 305.463,Z 456.057,A -85,B 0,C 180,E1 -16074.888,E2 -16074.888} C_VEL
LIN {X 0,Y 305.453,Z 456.06,A -85,B 0,C 180,E1 -16078.355,E2 -16078.355} C_VEL
LIN {X 0,Y 305.53,Z 456.049,A -85,B 0,C 180,E1 -16081.115,E2 -16081.115} C_VEL
LIN {X 0,Y 305.574,Z 456.045,A -85,B 0,C 180,E1 -16084.089,E2 -16084.089} C_VEL
LIN {X 0,Y 305.503,Z 456.053,A -85,B 0,C 180,E1 -16088.403,E2 -16088.403} C_VEL
LIN {X 0,Y 305.593,Z 456.043,A -85,B 0,C 180,E1 -16091.218,E2 -16091.218} C_VEL
LIN {X 0,Y 305.652,Z 456.037,A -85,B 0,C 180,E1 -16095.349,E2 -16095.349} C_VEL
LIN {X 0,Y 305.639,Z 456.039,A -85,B 0,C 180,E1 -16099.4,E2 -16099.4} C_VEL
LIN {X 0,Y 305.755,Z 456.022,A -85,B 0,C 180,E1 -16102.073,E2 -16102.073} C_VEL
LIN {X 0,Y 305.678,Z 456.031,A -85,B 0,C 180,E1 -16104.723,E2 -16104.723} C_VEL
LIN {X 0,Y 305.959,Z 455.995,A -85,B 0,C 180,E1 -16108.684,E2 -16108.684} C_VEL
LIN {X 0,Y 305.959,Z 456,A -85,B 0,C 180,E1 -16111.316,E2 -16111.316} C_VEL
LIN {X 0,Y 305.689,Z 456.034,A -85,B 0,C 180,E1 -16115.276,E2 -16115.276} C_VEL
LIN {X 0,Y 305.799,Z 456.016,A -85,B 0,C 180,E1 -16117.926,E2 -16117.926} C_VEL
LIN {X 0,Y 305.607,Z 456.04,A -85,B 0,C 180,E1 -16121.945,E2 -16121.945} C_VEL
LIN {X 0,Y 305.641,Z 456.039,A -85,B 0,C 180,E1 -16125.035,E2 -16125.035} C_VEL
LIN {X 0,Y 305.579,Z 456.046,A -85,B 0,C 180,E1 -16129.445,E2 -16129.445} C_VEL
LIN {X 0,Y 305.493,Z 456.059,A -85,B 0,C 180,E1 -16133.041,E2 -16133.041} C_VEL
LIN {X 0,Y 305.549,Z 456.047,A -85,B 0,C 180,E1 -16136.226,E2 -16136.226} C_VEL
LIN {X 0,Y 305.497,Z 456.058,A -85,B 0,C 180,E1 -16139.049,E2 -16139.049} C_VEL
LIN {X 0,Y 305.431,Z 456.061,A -85,B 0,C 180,E1 -16141.953,E2 -16141.953} C_VEL
LIN {X 0,Y 305.278,Z 456.084,A -85,B 0,C 180,E1 -16145.137,E2 -16145.137} C_VEL
LIN {X 0,Y 304.943,Z 456.124,A -85,B 0,C 180,E1 -16148.481,E2 -16148.481} C_VEL
LIN {X 0,Y 304.455,Z 456.188,A -85,B 0,C 180,E1 -16152.38,E2 -16152.38} C_VEL
LIN {X 0,Y 304.359,Z 457.947,A -85,B 0,C 180,E1 -16155.082,E2 -16155.082} C_VEL
LIN {X 0,Y 309.226,Z 475.159,A -85,B 0,C 180,E1 -16156.29,E2 -16156.29} C_VEL
LIN {X 0,Y 312.694,Z 488.56,A -85,B 0,C 180,E1 -16157.445,E2 -16157.445} C_VEL
LIN {X 0,Y 314.815,Z 497.984,A -85,B 0,C 180,E1 -16158.383,E2 -16158.383} C_VEL
LIN {X 0,Y 313.416,Z 511.287,A -85,B 0,C 180,E1 -16159.676,E2 -16159.676} C_VEL
LIN {X 0,Y 311.683,Z 524.412,A -85,B 0,C 180,E1 -16161.264,E2 -16161.264} C_VEL
LIN {X 0,Y 310.01,Z 536.478,A -85,B 0,C 180,E1 -16163.075,E2 -16163.075} C_VEL
LIN {X 0,Y 308.438,Z 547.564,A -85,B 0,C 180,E1 -16165.112,E2 -16165.112} C_VEL
LIN {X 0,Y 307.084,Z 556.337,A -85,B 0,C 180,E1 -16167.067,E2 -16167.067} C_VEL
LIN {X 0,Y 305.978,Z 564.467,A -85,B 0,C 180,E1 -16169.265,E2 -16169.265} C_VEL
LIN {X 0,Y 305.303,Z 570.014,A -85,B 0,C 180,E1 -16171.091,E2 -16171.091} C_VEL
LIN {X 0,Y 304.618,Z 575.484,A -85,B 0,C 180,E1 -16173.263,E2 -16173.263} C_VEL
LIN {X 0,Y 304.177,Z 579.8,A -85,B 0,C 180,E1 -16175.424,E2 -16175.424} C_VEL
LIN {X 0,Y 303.828,Z 583.242,A -85,B 0,C 180,E1 -16177.705,E2 -16177.705} C_VEL
LIN {X 0,Y 303.66,Z 585.354,A -85,B 0,C 180,E1 -16179.686,E2 -16179.686} C_VEL
LIN {X 0,Y 303.654,Z 586.645,A -85,B 0,C 180,E1 -16181.608,E2 -16181.608} C_VEL
LIN {X 0,Y 303.757,Z 587.285,A -85,B 0,C 180,E1 -16183.88,E2 -16183.88} C_VEL
LIN {X 0,Y 304.129,Z 586.705,A -85,B 0,C 180,E1 -16186.639,E2 -16186.639} C_VEL
LIN {X 0,Y 304.224,Z 586.322,A -85,B 0,C 180,E1 -16187.282,E2 -16187.282} C_VEL
LIN {X 0,Y 303.804,Z 585.689,A -85,B 0,C 180,E1 -16188.384,E2 -16188.384} C_VEL
LIN {X 0,Y 301.504,Z 584.313,A -85,B 0,C 180,E1 -16190.192,E2 -16190.192} C_VEL
LIN {X 0,Y 299.65,Z 582.869,A -85,B 0,C 180,E1 -16191.641,E2 -16191.641} C_VEL
LIN {X 0,Y 299.086,Z 581.452,A -85,B 0,C 180,E1 -16192.738,E2 -16192.738} C_VEL
LIN {X 0,Y 299.166,Z 580.87,A -85,B 0,C 180,E1 -16193.101,E2 -16193.101} C_VEL
LIN {X 0,Y 300.448,Z 576.816,A -85,B 0,C 180,E1 -16195.304,E2 -16195.304} C_VEL
LIN {X 0,Y 302.402,Z 570.516,A -85,B 0,C 180,E1 -16197.899,E2 -16197.899} C_VEL
LIN {X 0,Y 304.632,Z 563.04,A -85,B 0,C 180,E1 -16200.33,E2 -16200.33} C_VEL
LIN {X 0,Y 307.299,Z 554.183,A -85,B 0,C 180,E1 -16202.621,E2 -16202.621} C_VEL
LIN {X 0,Y 309.942,Z 544.984,A -85,B 0,C 180,E1 -16204.552,E2 -16204.552} C_VEL
LIN {X 0,Y 312.883,Z 534.089,A -85,B 0,C 180,E1 -16206.448,E2 -16206.448} C_VEL
LIN {X 0,Y 315.823,Z 521.933,A -85,B 0,C 180,E1 -16208.155,E2 -16208.155} C_VEL
LIN {X 0,Y 318.084,Z 511.78,A -85,B 0,C 180,E1 -16209.328,E2 -16209.328} C_VEL
LIN {X 0,Y 317.381,Z 506.136,A -85,B 0,C 180,E1 -16210.204,E2 -16210.204} C_VEL
LIN {X 0,Y 315.154,Z 498.102,A -85,B 0,C 180,E1 -16211.578,E2 -16211.578} C_VEL
LIN {X 0,Y 310.895,Z 487.435,A -85,B 0,C 180,E1 -16213.584,E2 -16213.584} C_VEL
LIN {X 0,Y 305.174,Z 476.359,A -85,B 0,C 180,E1 -16215.943,E2 -16215.943} C_VEL
LIN {X 0,Y 303.156,Z 473.325,A -85,B 0,C 180,E1 -16216.723,E2 -16216.723} C_VEL
LIN {X 0,Y 302.494,Z 471.954,A -85,B 0,C 180,E1 -16217.024,E2 -16217.024} C_VEL
LIN {X 0,Y 300.413,Z 469.432,A -85,B 0,C 180,E1 -16217.793,E2 -16217.793} C_VEL
LIN {X 0,Y 299.669,Z 467.215,A -85,B 0,C 180,E1 -16218.192,E2 -16218.192} C_VEL
LIN {X 0,Y 299.856,Z 466.779,A -85,B 0,C 180,E1 -16220.583,E2 -16220.583} C_VEL
LIN {X 0,Y 299.984,Z 466.466,A -85,B 0,C 180,E1 -16223.982,E2 -16223.982} C_VEL
LIN {X 0,Y 300.054,Z 466.584,A -85,B 0,C 180,E1 -16227.933,E2 -16227.933} C_VEL
LIN {X 0,Y 300.171,Z 467.042,A -85,B 0,C 180,E1 -16231.003,E2 -16231.003} C_VEL
LIN {X 0,Y 300.385,Z 468.199,A -85,B 0,C 180,E1 -16235.028,E2 -16235.028} C_VEL
LIN {X 0,Y 300.733,Z 470.044,A -85,B 0,C 180,E1 -16239.122,E2 -16239.122} C_VEL
LIN {X 0,Y 301.104,Z 472.18,A -85,B 0,C 180,E1 -16242.6,E2 -16242.6} C_VEL
LIN {X 0,Y 301.546,Z 474.979,A -85,B 0,C 180,E1 -16246.261,E2 -16246.261} C_VEL
LIN {X 0,Y 301.676,Z 477.803,A -85,B 0,C 180,E1 -16249.286,E2 -16249.286} C_VEL
LIN {X 0,Y 301.541,Z 479.609,A -85,B 0,C 180,E1 -16251.003,E2 -16251.003} C_VEL
LIN {X 0,Y 300.839,Z 483.158,A -85,B 0,C 180,E1 -16254.034,E2 -16254.034} C_VEL
LIN {X 0,Y 301.769,Z 486.65,A -85,B 0,C 180,E1 -16254.549,E2 -16254.549} C_VEL
LIN {X 0,Y 303.18,Z 489.287,A -85,B 0,C 180,E1 -16255.093,E2 -16255.093} C_VEL
LIN {X 0,Y 304.692,Z 493.49,A -85,B 0,C 180,E1 -16255.769,E2 -16255.769} C_VEL
LIN {X 0,Y 307.756,Z 502.62,A -85,B 0,C 180,E1 -16257.21,E2 -16257.21} C_VEL
LIN {X 0,Y 310.727,Z 514.098,A -85,B 0,C 180,E1 -16258.872,E2 -16258.872} C_VEL
LIN {X 0,Y 312.722,Z 526.582,A -85,B 0,C 180,E1 -16260.558,E2 -16260.558} C_VEL
LIN {X 0,Y 313.383,Z 536.646,A -85,B 0,C 180,E1 -16261.904,E2 -16261.904} C_VEL
LIN {X 0,Y 313.07,Z 547.209,A -85,B 0,C 180,E1 -16263.323,E2 -16263.323} C_VEL
LIN {X 0,Y 312.384,Z 552.102,A -85,B 0,C 180,E1 -16263.979,E2 -16263.979} C_VEL
LIN {X 0,Y 309.419,Z 563.588,A -85,B 0,C 180,E1 -16265.573,E2 -16265.573} C_VEL
LIN {X 0,Y 306.57,Z 574.575,A -85,B 0,C 180,E1 -16267.42,E2 -16267.42} C_VEL
LIN {X 0,Y 304.071,Z 584.106,A -85,B 0,C 180,E1 -16269.362,E2 -16269.362} C_VEL
LIN {X 0,Y 301.638,Z 593.427,A -85,B 0,C 180,E1 -16271.667,E2 -16271.667} C_VEL
LIN {X 0,Y 299.698,Z 601.281,A -85,B 0,C 180,E1 -16274.041,E2 -16274.041} C_VEL
LIN {X 0,Y 298.427,Z 607.494,A -85,B 0,C 180,E1 -16276.379,E2 -16276.379} C_VEL
LIN {X 0,Y 297.282,Z 613.173,A -85,B 0,C 180,E1 -16279.098,E2 -16279.098} C_VEL
LIN {X 0,Y 296.785,Z 617.357,A -85,B 0,C 180,E1 -16281.832,E2 -16281.832} C_VEL
LIN {X 0,Y 296.599,Z 620.122,A -85,B 0,C 180,E1 -16284.561,E2 -16284.561} C_VEL
LIN {X 0,Y 296.663,Z 621.504,A -85,B 0,C 180,E1 -16287.284,E2 -16287.284} C_VEL
LIN {X 0,Y 296.946,Z 621.5,A -85,B 0,C 180,E1 -16290,E2 -16290} C_VEL
LIN {X 0,Y 296.835,Z 620.947,A -85,B 0,C 180,E1 -16291.357,E2 -16291.357} C_VEL
LIN {X 0,Y 296.735,Z 618.757,A -85,B 0,C 180,E1 -16294.074,E2 -16294.074} C_VEL
LIN {X 0,Y 296.784,Z 616.365,A -85,B 0,C 180,E1 -16295.967,E2 -16295.967} C_VEL
LIN {X 0,Y 296.868,Z 612.617,A -85,B 0,C 180,E1 -16298.166,E2 -16298.166} C_VEL
LIN {X 0,Y 297.144,Z 608.095,A -85,B 0,C 180,E1 -16300.218,E2 -16300.218} C_VEL
LIN {X 0,Y 297.847,Z 601.545,A -85,B 0,C 180,E1 -16302.607,E2 -16302.607} C_VEL
LIN {X 0,Y 298.542,Z 594.605,A -85,B 0,C 180,E1 -16304.659,E2 -16304.659} C_VEL
LIN {X 0,Y 299.738,Z 586.317,A -85,B 0,C 180,E1 -16306.692,E2 -16306.692} C_VEL
LIN {X 0,Y 301.206,Z 576.364,A -85,B 0,C 180,E1 -16308.713,E2 -16308.713} C_VEL
LIN {X 0,Y 302.886,Z 565.386,A -85,B 0,C 180,E1 -16310.545,E2 -16310.545} C_VEL
LIN {X 0,Y 304.761,Z 553.283,A -85,B 0,C 180,E1 -16312.186,E2 -16312.186} C_VEL
LIN {X 0,Y 305.928,Z 543.114,A -85,B 0,C 180,E1 -16313.345,E2 -16313.345} C_VEL
LIN {X 0,Y 304.502,Z 529.745,A -85,B 0,C 180,E1 -16314.73,E2 -16314.73} C_VEL
LIN {X 0,Y 302.447,Z 514.973,A -85,B 0,C 180,E1 -16315.994,E2 -16315.994} C_VEL
LIN {X 0,Y 299.951,Z 499.844,A -85,B 0,C 180,E1 -16317.033,E2 -16317.033} C_VEL
LIN {X 0,Y 298.39,Z 491.172,A -85,B 0,C 180,E1 -16317.545,E2 -16317.545} C_VEL
LIN {X 0,Y 299.147,Z 485.605,A -85,B 0,C 180,E1 -16321.121,E2 -16321.121} C_VEL
LIN {X 0,Y 300.033,Z 479.784,A -85,B 0,C 180,E1 -16324.931,E2 -16324.931} C_VEL
LIN {X 0,Y 300.802,Z 474.839,A -85,B 0,C 180,E1 -16328.253,E2 -16328.253} C_VEL
LIN {X 0,Y 300.992,Z 472.896,A -85,B 0,C 180,E1 -16329.599,E2 -16329.599} C_VEL
LIN {X 0,Y 300.767,Z 470.117,A -85,B 0,C 180,E1 -16331.605,E2 -16331.605} C_VEL
LIN {X 0,Y 299.917,Z 465.183,A -85,B 0,C 180,E1 -16335.333,E2 -16335.333} C_VEL
LIN {X 0,Y 298.953,Z 459.703,A -85,B 0,C 180,E1 -16339.723,E2 -16339.723} C_VEL
LIN {X 0,Y 298.489,Z 456.932,A -85,B 0,C 180,E1 -16342.253,E2 -16342.253} C_VEL
LIN {X 0,Y 298.405,Z 456.937,A -85,B 0,C 180,E1 -16345.581,E2 -16345.581} C_VEL
LIN {X 0,Y 298.395,Z 456.941,A -85,B 0,C 180,E1 -16348.791,E2 -16348.791} C_VEL
LIN {X 0,Y 298.46,Z 456.93,A -85,B 0,C 180,E1 -16351.904,E2 -16351.904} C_VEL
LIN {X 0,Y 298.481,Z 456.931,A -85,B 0,C 180,E1 -16354.924,E2 -16354.924} C_VEL
LIN {X 0,Y 298.446,Z 456.933,A -85,B 0,C 180,E1 -16359.315,E2 -16359.315} C_VEL
LIN {X 0,Y 298.533,Z 456.921,A -85,B 0,C 180,E1 -16362.179,E2 -16362.179} C_VEL
LIN {X 0,Y 298.589,Z 456.917,A -85,B 0,C 180,E1 -16364.995,E2 -16364.995} C_VEL
LIN {X 0,Y 298.589,Z 456.916,A -85,B 0,C 180,E1 -16369.147,E2 -16369.147} C_VEL
LIN {X 0,Y 298.753,Z 456.893,A -85,B 0,C 180,E1 -16371.886,E2 -16371.886} C_VEL
LIN {X 0,Y 298.656,Z 456.909,A -85,B 0,C 180,E1 -16374.599,E2 -16374.599} C_VEL
LIN {X 0,Y 298.92,Z 456.877,A -85,B 0,C 180,E1 -16378.653,E2 -16378.653} C_VEL
LIN {X 0,Y 298.921,Z 456.872,A -85,B 0,C 180,E1 -16381.347,E2 -16381.347} C_VEL
LIN {X 0,Y 298.659,Z 456.905,A -85,B 0,C 180,E1 -16385.401,E2 -16385.401} C_VEL
LIN {X 0,Y 298.755,Z 456.895,A -85,B 0,C 180,E1 -16388.114,E2 -16388.114} C_VEL
LIN {X 0,Y 298.549,Z 456.921,A -85,B 0,C 180,E1 -16392.232,E2 -16392.232} C_VEL
LIN {X 0,Y 298.581,Z 456.915,A -85,B 0,C 180,E1 -16395.195,E2 -16395.195} C_VEL
LIN {X 0,Y 298.536,Z 456.919,A -85,B 0,C 180,E1 -16399.244,E2 -16399.244} C_VEL
LIN {X 0,Y 298.454,Z 456.931,A -85,B 0,C 180,E1 -16403.598,E2 -16403.598} C_VEL
LIN {X 0,Y 298.486,Z 456.928,A -85,B 0,C 180,E1 -16406.575,E2 -16406.575} C_VEL
LIN {X 0,Y 298.418,Z 456.935,A -85,B 0,C 180,E1 -16409.642,E2 -16409.642} C_VEL
LIN {X 0,Y 298.393,Z 456.939,A -85,B 0,C 180,E1 -16412.801,E2 -16412.801} C_VEL
LIN {X 0,Y 298.444,Z 456.931,A -85,B 0,C 180,E1 -16416.808,E2 -16416.808} C_VEL
LIN {X 0,Y 298.407,Z 456.937,A -85,B 0,C 180,E1 -16419.487,E2 -16419.487} C_VEL
LIN {X 0,Y 298.397,Z 456.937,A -85,B 0,C 180,E1 -16423.104,E2 -16423.104} C_VEL
LIN {X 0,Y 298.431,Z 456.933,A -85,B 0,C 180,E1 -16426.927,E2 -16426.927} C_VEL
LIN {X 0,Y 298.431,Z 456.933,A -85,B 0,C 180,E1 -16431,E2 -16431} C_VEL
LIN {X 0,Y 298.433,Z 456.937,A -85,B 0,C 180,E1 -16433.933,E2 -16433.933} C_VEL
LIN {X 0,Y 298.397,Z 456.941,A -85,B 0,C 180,E1 -16437.984,E2 -16437.984} C_VEL
LIN {X 0,Y 298.478,Z 456.931,A -85,B 0,C 180,E1 -16441.906,E2 -16441.906} C_VEL
LIN {X 0,Y 298.488,Z 456.926,A -85,B 0,C 180,E1 -16444.925,E2 -16444.925} C_VEL
LIN {X 0,Y 298.453,Z 456.933,A -85,B 0,C 180,E1 -16449.316,E2 -16449.316} C_VEL
LIN {X 0,Y 298.54,Z 456.92,A -85,B 0,C 180,E1 -16452.18,E2 -16452.18} C_VEL
LIN {X 0,Y 298.596,Z 456.913,A -85,B 0,C 180,E1 -16454.995,E2 -16454.995} C_VEL
LIN {X 0,Y 298.595,Z 456.915,A -85,B 0,C 180,E1 -16459.147,E2 -16459.147} C_VEL
LIN {X 0,Y 298.705,Z 456.901,A -85,B 0,C 180,E1 -16461.885,E2 -16461.885} C_VEL
LIN {X 0,Y 298.647,Z 456.906,A -85,B 0,C 180,E1 -16464.599,E2 -16464.599} C_VEL
LIN {X 0,Y 298.926,Z 456.871,A -85,B 0,C 180,E1 -16468.653,E2 -16468.653} C_VEL
LIN {X 0,Y 298.926,Z 456.876,A -85,B 0,C 180,E1 -16471.347,E2 -16471.347} C_VEL
LIN {X 0,Y 298.79,Z 456.889,A -85,B 0,C 180,E1 -16476.754,E2 -16476.754} C_VEL
LIN {X 0,Y 298.639,Z 456.91,A -85,B 0,C 180,E1 -16479.482,E2 -16479.482} C_VEL
LIN {X 0,Y 298.556,Z 456.92,A -85,B 0,C 180,E1 -16483.615,E2 -16483.615} C_VEL
LIN {X 0,Y 298.552,Z 456.919,A -85,B 0,C 180,E1 -16486.408,E2 -16486.408} C_VEL
LIN {X 0,Y 298.514,Z 456.924,A -85,B 0,C 180,E1 -16489.654,E2 -16489.654} C_VEL
LIN {X 0,Y 298.46,Z 456.931,A -85,B 0,C 180,E1 -16493.597,E2 -16493.597} C_VEL
LIN {X 0,Y 298.491,Z 456.927,A -85,B 0,C 180,E1 -16496.574,E2 -16496.574} C_VEL
LIN {X 0,Y 298.422,Z 456.935,A -85,B 0,C 180,E1 -16499.64,E2 -16499.64} C_VEL
LIN {X 0,Y 298.352,Z 456.947,A -85,B 0,C 180,E1 -16502.805,E2 -16502.805} C_VEL
LIN {X 0,Y 298.146,Z 456.969,A -85,B 0,C 180,E1 -16506.107,E2 -16506.107} C_VEL
LIN {X 0,Y 297.749,Z 457.024,A -85,B 0,C 180,E1 -16509.59,E2 -16509.59} C_VEL
LIN {X 0,Y 297.334,Z 457.075,A -85,B 0,C 180,E1 -16512.883,E2 -16512.883} C_VEL
LIN {X 0,Y 297.312,Z 458.317,A -85,B 0,C 180,E1 -16514.595,E2 -16514.595} C_VEL
LIN {X 0,Y 301.915,Z 474.432,A -85,B 0,C 180,E1 -16515.755,E2 -16515.755} C_VEL
LIN {X 0,Y 305.401,Z 488.005,A -85,B 0,C 180,E1 -16516.941,E2 -16516.941} C_VEL
LIN {X 0,Y 307.81,Z 498.597,A -85,B 0,C 180,E1 -16518.021,E2 -16518.021} C_VEL
LIN {X 0,Y 307.968,Z 500.127,A -85,B 0,C 180,E1 -16518.174,E2 -16518.174} C_VEL
LIN {X 0,Y 306.362,Z 513.403,A -85,B 0,C 180,E1 -16519.529,E2 -16519.529} C_VEL
LIN {X 0,Y 304.716,Z 525.517,A -85,B 0,C 180,E1 -16521.06,E2 -16521.06} C_VEL
LIN {X 0,Y 302.966,Z 537.448,A -85,B 0,C 180,E1 -16522.905,E2 -16522.905} C_VEL
LIN {X 0,Y 301.463,Z 547.975,A -85,B 0,C 180,E1 -16524.893,E2 -16524.893} C_VEL
LIN {X 0,Y 299.991,Z 557.184,A -85,B 0,C 180,E1 -16526.996,E2 -16526.996} C_VEL
LIN {X 0,Y 298.878,Z 565.213,A -85,B 0,C 180,E1 -16529.24,E2 -16529.24} C_VEL
LIN {X 0,Y 298.16,Z 571.107,A -85,B 0,C 180,E1 -16531.249,E2 -16531.249} C_VEL
LIN {X 0,Y 297.395,Z 577.36,A -85,B 0,C 180,E1 -16533.896,E2 -16533.896} C_VEL
LIN {X 0,Y 296.932,Z 581.619,A -85,B 0,C 180,E1 -16536.273,E2 -16536.273} C_VEL
LIN {X 0,Y 296.754,Z 583.627,A -85,B 0,C 180,E1 -16537.732,E2 -16537.732} C_VEL
LIN {X 0,Y 296.524,Z 586.407,A -85,B 0,C 180,E1 -16540.621,E2 -16540.621} C_VEL
LIN {X 0,Y 296.572,Z 587.217,A -85,B 0,C 180,E1 -16542.057,E2 -16542.057} C_VEL
LIN {X 0,Y 296.77,Z 587.726,A -85,B 0,C 180,E1 -16544.9,E2 -16544.9} C_VEL
LIN {X 0,Y 297.251,Z 586.792,A -85,B 0,C 180,E1 -16547.714,E2 -16547.714} C_VEL
LIN {X 0,Y 298.047,Z 584.425,A -85,B 0,C 180,E1 -16550.499,E2 -16550.499} C_VEL
LIN {X 0,Y 299.166,Z 580.87,A -85,B 0,C 180,E1 -16553.101,E2 -16553.101} C_VEL
LIN {X 0,Y 299.06,Z 579.178,A -85,B 0,C 180,E1 -16554.186,E2 -16554.186} C_VEL
LIN {X 0,Y 297.361,Z 576.268,A -85,B 0,C 180,E1 -16555.98,E2 -16555.98} C_VEL
LIN {X 0,Y 296.051,Z 573.57,A -85,B 0,C 180,E1 -16557.4,E2 -16557.4} C_VEL
LIN {X 0,Y 295.912,Z 571.166,A -85,B 0,C 180,E1 -16558.443,E2 -16558.443} C_VEL
LIN {X 0,Y 296.133,Z 570.261,A -85,B 0,C 180,E1 -16558.78,E2 -16558.78} C_VEL
LIN {X 0,Y 298.705,Z 562.294,A -85,B 0,C 180,E1 -16561.348,E2 -16561.348} C_VEL
